LIN {X 0,Y 468.258,Z 232.885,A -85,B 0,C 180,E1 -7689.078,E2 -7689.078} C_VEL
LIN {X 0,Y 467.789,Z 228.961,A -85,B 0,C 180,E1 -7691.38,E2 -7691.38} C_VEL
LIN {X 0,Y 467.563,Z 227.872,A -85,B 0,C 180,E1 -7692.126,E2 -7692.126} C_VEL
LIN {X 0,Y 467.566,Z 227.872,A -85,B 0,C 180,E1 -7695.053,E2 -7695.053} C_VEL
LIN {X 0,Y 467.59,Z 227.868,A -85,B 0,C 180,E1 -7697.44,E2 -7697.44} C_VEL
LIN {X 0,Y 467.576,Z 227.87,A -85,B 0,C 180,E1 -7700.855,E2 -7700.855} C_VEL
LIN {X 0,Y 467.558,Z 227.874,A -85,B 0,C 180,E1 -7704.261,E2 -7704.261} C_VEL
LIN {X 0,Y 467.583,Z 227.869,A -85,B 0,C 180,E1 -7707.321,E2 -7707.321} C_VEL
LIN {X 0,Y 467.554,Z 227.872,A -85,B 0,C 180,E1 -7710.671,E2 -7710.671} C_VEL
LIN {X 0,Y 467.559,Z 227.867,A -85,B 0,C 180,E1 -7713.196,E2 -7713.196} C_VEL
LIN {X 0,Y 467.591,Z 227.864,A -85,B 0,C 180,E1 -7716.469,E2 -7716.469} C_VEL
LIN {X 0,Y 467.622,Z 227.86,A -85,B 0,C 180,E1 -7719.777,E2 -7719.777} C_VEL
LIN {X 0,Y 467.591,Z 227.864,A -85,B 0,C 180,E1 -7722.506,E2 -7722.506} C_VEL
LIN {X 0,Y 467.611,Z 227.864,A -85,B 0,C 180,E1 -7725.197,E2 -7725.197} C_VEL
LIN {X 0,Y 467.658,Z 227.855,A -85,B 0,C 180,E1 -7727.855,E2 -7727.855} C_VEL
LIN {X 0,Y 467.659,Z 227.855,A -85,B 0,C 180,E1 -7731.357,E2 -7731.357} C_VEL
LIN {X 0,Y 467.713,Z 227.849,A -85,B 0,C 180,E1 -7733.962,E2 -7733.962} C_VEL
LIN {X 0,Y 467.861,Z 227.83,A -85,B 0,C 180,E1 -7737.417,E2 -7737.417} C_VEL
LIN {X 0,Y 467.88,Z 227.832,A -85,B 0,C 180,E1 -7740,E2 -7740} C_VEL
LIN {X 0,Y 467.849,Z 227.831,A -85,B 0,C 180,E1 -7742.583,E2 -7742.583} C_VEL
LIN {X 0,Y 467.737,Z 227.846,A -85,B 0,C 180,E1 -7746.038,E2 -7746.038} C_VEL
LIN {X 0,Y 467.682,Z 227.852,A -85,B 0,C 180,E1 -7748.643,E2 -7748.643} C_VEL
LIN {X 0,Y 467.656,Z 227.855,A -85,B 0,C 180,E1 -7752.358,E2 -7752.358} C_VEL
LIN {X 0,Y 467.652,Z 227.858,A -85,B 0,C 180,E1 -7755.885,E2 -7755.885} C_VEL
LIN {X 0,Y 467.625,Z 227.863,A -85,B 0,C 180,E1 -7759.308,E2 -7759.308} C_VEL
LIN {X 0,Y 467.536,Z 227.87,A -85,B 0,C 180,E1 -7762.074,E2 -7762.074} C_VEL
LIN {X 0,Y 467.587,Z 227.864,A -85,B 0,C 180,E1 -7764.888,E2 -7764.888} C_VEL
LIN {X 0,Y 467.621,Z 227.863,A -85,B 0,C 180,E1 -7767.769,E2 -7767.769} C_VEL
LIN {X 0,Y 467.569,Z 227.869,A -85,B 0,C 180,E1 -7771.045,E2 -7771.045} C_VEL
LIN {X 0,Y 467.579,Z 227.868,A -85,B 0,C 180,E1 -7774.24,E2 -7774.24} C_VEL
LIN {X 0,Y 467.549,Z 227.873,A -85,B 0,C 180,E1 -7777.186,E2 -7777.186} C_VEL
LIN {X 0,Y 467.56,Z 227.869,A -85,B 0,C 180,E1 -7780.267,E2 -7780.267} C_VEL
LIN {X 0,Y 467.549,Z 227.874,A -85,B 0,C 180,E1 -7783.745,E2 -7783.745} C_VEL
LIN {X 0,Y 467.556,Z 227.869,A -85,B 0,C 180,E1 -7786.255,E2 -7786.255} C_VEL
LIN {X 0,Y 467.572,Z 227.872,A -85,B 0,C 180,E1 -7788.724,E2 -7788.724} C_VEL
LIN {X 0,Y 467.563,Z 227.872,A -85,B 0,C 180,E1 -7790.049,E2 -7790.049} C_VEL
LIN {X 0,Y 467.556,Z 228.203,A -85,B 0,C 180,E1 -7790.853,E2 -7790.853} C_VEL
LIN {X 0,Y 467.607,Z 231.102,A -85,B 0,C 180,E1 -7793.045,E2 -7793.045} C_VEL
LIN {X 0,Y 467.545,Z 234.837,A -85,B 0,C 180,E1 -7795.766,E2 -7795.766} C_VEL
LIN {X 0,Y 467.357,Z 239.771,A -85,B 0,C 180,E1 -7799.251,E2 -7799.251} C_VEL
LIN {X 0,Y 467.155,Z 244.635,A -85,B 0,C 180,E1 -7802.575,E2 -7802.575} C_VEL
LIN {X 0,Y 467.087,Z 248.387,A -85,B 0,C 180,E1 -7805.083,E2 -7805.083} C_VEL
LIN {X 0,Y 466.975,Z 252.771,A -85,B 0,C 180,E1 -7807.898,E2 -7807.898} C_VEL
LIN {X 0,Y 466.904,Z 258.071,A -85,B 0,C 180,E1 -7811.245,E2 -7811.245} C_VEL
LIN {X 0,Y 466.903,Z 258.381,A -85,B 0,C 180,E1 -7811.432,E2 -7811.432} C_VEL
LIN {X 0,Y 470.586,Z 273.156,A -85,B 0,C 180,E1 -7811.948,E2 -7811.948} C_VEL
LIN {X 0,Y 471.87,Z 279.673,A -85,B 0,C 180,E1 -7812.223,E2 -7812.223} C_VEL
LIN {X 0,Y 471.651,Z 287.48,A -85,B 0,C 180,E1 -7812.533,E2 -7812.533} C_VEL
LIN {X 0,Y 470.858,Z 293.031,A -85,B 0,C 180,E1 -7812.76,E2 -7812.76} C_VEL
LIN {X 0,Y 467.715,Z 301.937,A -85,B 0,C 180,E1 -7813.131,E2 -7813.131} C_VEL
LIN {X 0,Y 464.47,Z 310.546,A -85,B 0,C 180,E1 -7813.583,E2 -7813.583} C_VEL
LIN {X 0,Y 463.524,Z 315.627,A -85,B 0,C 180,E1 -7813.933,E2 -7813.933} C_VEL
LIN {X 0,Y 462.813,Z 327.365,A -85,B 0,C 180,E1 -7814.927,E2 -7814.927} C_VEL
LIN {X 0,Y 462.041,Z 339.043,A -85,B 0,C 180,E1 -7816.139,E2 -7816.139} C_VEL
LIN {X 0,Y 461.354,Z 349.678,A -85,B 0,C 180,E1 -7817.491,E2 -7817.491} C_VEL
LIN {X 0,Y 460.845,Z 358.072,A -85,B 0,C 180,E1 -7818.788,E2 -7818.788} C_VEL
LIN {X 0,Y 460.359,Z 366.316,A -85,B 0,C 180,E1 -7820.333,E2 -7820.333} C_VEL
LIN {X 0,Y 460.082,Z 372.056,A -85,B 0,C 180,E1 -7821.656,E2 -7821.656} C_VEL
LIN {X 0,Y 459.847,Z 376.778,A -85,B 0,C 180,E1 -7822.977,E2 -7822.977} C_VEL
LIN {X 0,Y 459.728,Z 381.668,A -85,B 0,C 180,E1 -7824.737,E2 -7824.737} C_VEL
LIN {X 0,Y 459.623,Z 385.073,A -85,B 0,C 180,E1 -7826.493,E2 -7826.493} C_VEL
LIN {X 0,Y 459.519,Z 387.099,A -85,B 0,C 180,E1 -7828.247,E2 -7828.247} C_VEL
LIN {X 0,Y 459.5,Z 387.796,A -85,B 0,C 180,E1 -7830,E2 -7830} C_VEL
LIN {X 0,Y 459.518,Z 387.175,A -85,B 0,C 180,E1 -7831.753,E2 -7831.753} C_VEL
LIN {X 0,Y 459.622,Z 385.219,A -85,B 0,C 180,E1 -7833.507,E2 -7833.507} C_VEL
LIN {X 0,Y 459.722,Z 381.883,A -85,B 0,C 180,E1 -7835.263,E2 -7835.263} C_VEL
LIN {X 0,Y 459.847,Z 377.072,A -85,B 0,C 180,E1 -7837.023,E2 -7837.023} C_VEL
LIN {X 0,Y 460.134,Z 370.627,A -85,B 0,C 180,E1 -7838.786,E2 -7838.786} C_VEL
LIN {X 0,Y 460.502,Z 363.45,A -85,B 0,C 180,E1 -7840.331,E2 -7840.331} C_VEL
LIN {X 0,Y 461.108,Z 354.57,A -85,B 0,C 180,E1 -7841.874,E2 -7841.874} C_VEL
LIN {X 0,Y 461.665,Z 345.24,A -85,B 0,C 180,E1 -7843.2,E2 -7843.2} C_VEL
LIN {X 0,Y 462.317,Z 334.904,A -85,B 0,C 180,E1 -7844.414,E2 -7844.414} C_VEL
LIN {X 0,Y 463.038,Z 323.496,A -85,B 0,C 180,E1 -7845.516,E2 -7845.516} C_VEL
LIN {X 0,Y 463.776,Z 310.849,A -85,B 0,C 180,E1 -7846.507,E2 -7846.507} C_VEL
LIN {X 0,Y 464.402,Z 297.961,A -85,B 0,C 180,E1 -7847.311,E2 -7847.311} C_VEL
LIN {X 0,Y 464.97,Z 283.959,A -85,B 0,C 180,E1 -7847.979,E2 -7847.979} C_VEL
LIN {X 0,Y 464.881,Z 279.458,A -85,B 0,C 180,E1 -7848.16,E2 -7848.16} C_VEL
LIN {X 0,Y 461.702,Z 265.746,A -85,B 0,C 180,E1 -7848.721,E2 -7848.721} C_VEL
LIN {X 0,Y 459.856,Z 258.473,A -85,B 0,C 180,E1 -7848.975,E2 -7848.975} C_VEL
LIN {X 0,Y 459.938,Z 253.029,A -85,B 0,C 180,E1 -7852.458,E2 -7852.458} C_VEL
LIN {X 0,Y 460.035,Z 248.128,A -85,B 0,C 180,E1 -7855.664,E2 -7855.664} C_VEL
LIN {X 0,Y 460.143,Z 244.325,A -85,B 0,C 180,E1 -7858.261,E2 -7858.261} C_VEL
LIN {X 0,Y 460.332,Z 240.017,A -85,B 0,C 180,E1 -7861.271,E2 -7861.271} C_VEL
LIN {X 0,Y 460.526,Z 235.502,A -85,B 0,C 180,E1 -7864.504,E2 -7864.504} C_VEL
LIN {X 0,Y 460.553,Z 231.318,A -85,B 0,C 180,E1 -7867.618,E2 -7867.618} C_VEL
LIN {X 0,Y 460.542,Z 229.642,A -85,B 0,C 180,E1 -7868.897,E2 -7868.897} C_VEL
LIN {X 0,Y 460.491,Z 228.756,A -85,B 0,C 180,E1 -7869.867,E2 -7869.867} C_VEL
LIN {X 0,Y 460.516,Z 228.749,A -85,B 0,C 180,E1 -7872.901,E2 -7872.901} C_VEL
LIN {X 0,Y 460.51,Z 228.748,A -85,B 0,C 180,E1 -7875.831,E2 -7875.831} C_VEL
LIN {X 0,Y 460.521,Z 228.746,A -85,B 0,C 180,E1 -7878.987,E2 -7878.987} C_VEL
LIN {X 0,Y 460.517,Z 228.749,A -85,B 0,C 180,E1 -7881.266,E2 -7881.266} C_VEL
LIN {X 0,Y 460.511,Z 228.749,A -85,B 0,C 180,E1 -7884.554,E2 -7884.554} C_VEL
LIN {X 0,Y 460.532,Z 228.747,A -85,B 0,C 180,E1 -7887.716,E2 -7887.716} C_VEL
LIN {X 0,Y 460.54,Z 228.746,A -85,B 0,C 180,E1 -7890.769,E2 -7890.769} C_VEL
LIN {X 0,Y 460.559,Z 228.741,A -85,B 0,C 180,E1 -7893.734,E2 -7893.734} C_VEL
LIN {X 0,Y 460.548,Z 228.741,A -85,B 0,C 180,E1 -7896.624,E2 -7896.624} C_VEL
LIN {X 0,Y 460.554,Z 228.74,A -85,B 0,C 180,E1 -7899.453,E2 -7899.453} C_VEL
LIN {X 0,Y 460.551,Z 228.744,A -85,B 0,C 180,E1 -7902.23,E2 -7902.23} C_VEL
LIN {X 0,Y 460.567,Z 228.739,A -85,B 0,C 180,E1 -7904.965,E2 -7904.965} C_VEL
LIN {X 0,Y 460.613,Z 228.736,A -85,B 0,C 180,E1 -7908.559,E2 -7908.559} C_VEL
LIN {X 0,Y 460.622,Z 228.731,A -85,B 0,C 180,E1 -7911.224,E2 -7911.224} C_VEL
LIN {X 0,Y 460.703,Z 228.723,A -85,B 0,C 180,E1 -7913.87,E2 -7913.87} C_VEL
LIN {X 0,Y 460.792,Z 228.71,A -85,B 0,C 180,E1 -7917.377,E2 -7917.377} C_VEL
LIN {X 0,Y 460.825,Z 228.71,A -85,B 0,C 180,E1 -7920,E2 -7920} C_VEL
LIN {X 0,Y 460.803,Z 228.708,A -85,B 0,C 180,E1 -7922.622,E2 -7922.622} C_VEL
LIN {X 0,Y 460.679,Z 228.726,A -85,B 0,C 180,E1 -7926.13,E2 -7926.13} C_VEL
LIN {X 0,Y 460.612,Z 228.733,A -85,B 0,C 180,E1 -7928.776,E2 -7928.776} C_VEL
LIN {X 0,Y 460.617,Z 228.732,A -85,B 0,C 180,E1 -7932.445,E2 -7932.445} C_VEL
LIN {X 0,Y 460.604,Z 228.737,A -85,B 0,C 180,E1 -7935.997,E2 -7935.997} C_VEL
LIN {X 0,Y 460.569,Z 228.743,A -85,B 0,C 180,E1 -7939.615,E2 -7939.615} C_VEL
LIN {X 0,Y 460.514,Z 228.747,A -85,B 0,C 180,E1 -7942.428,E2 -7942.428} C_VEL
LIN {X 0,Y 460.546,Z 228.742,A -85,B 0,C 180,E1 -7945.796,E2 -7945.796} C_VEL
LIN {X 0,Y 460.522,Z 228.748,A -85,B 0,C 180,E1 -7949.232,E2 -7949.232} C_VEL
LIN {X 0,Y 460.534,Z 228.746,A -85,B 0,C 180,E1 -7952.284,E2 -7952.284} C_VEL
LIN {X 0,Y 460.51,Z 228.75,A -85,B 0,C 180,E1 -7955.446,E2 -7955.446} C_VEL
LIN {X 0,Y 460.542,Z 228.747,A -85,B 0,C 180,E1 -7958.897,E2 -7958.897} C_VEL
LIN {X 0,Y 460.525,Z 228.751,A -85,B 0,C 180,E1 -7962.181,E2 -7962.181} C_VEL
LIN {X 0,Y 460.513,Z 228.751,A -85,B 0,C 180,E1 -7965.411,E2 -7965.411} C_VEL
LIN {X 0,Y 460.558,Z 228.925,A -85,B 0,C 180,E1 -7967.822,E2 -7967.822} C_VEL
LIN {X 0,Y 461.132,Z 232.835,A -85,B 0,C 180,E1 -7970.2,E2 -7970.2} C_VEL
LIN {X 0,Y 461.314,Z 236.792,A -85,B 0,C 180,E1 -7972.454,E2 -7972.454} C_VEL
LIN {X 0,Y 461.036,Z 242.718,A -85,B 0,C 180,E1 -7975.665,E2 -7975.665} C_VEL
LIN {X 0,Y 460.839,Z 248.673,A -85,B 0,C 180,E1 -7978.767,E2 -7978.767} C_VEL
LIN {X 0,Y 460.613,Z 255.61,A -85,B 0,C 180,E1 -7982.247,E2 -7982.247} C_VEL
LIN {X 0,Y 460.218,Z 262.588,A -85,B 0,C 180,E1 -7985.649,E2 -7985.649} C_VEL
LIN {X 0,Y 460.068,Z 268.978,A -85,B 0,C 180,E1 -7988.723,E2 -7988.723} C_VEL
LIN {X 0,Y 459.911,Z 273.938,A -85,B 0,C 180,E1 -7991.062,E2 -7991.062} C_VEL
LIN {X 0,Y 463.398,Z 290.247,A -85,B 0,C 180,E1 -7991.618,E2 -7991.618} C_VEL
LIN {X 0,Y 464.84,Z 299.475,A -85,B 0,C 180,E1 -7992.006,E2 -7992.006} C_VEL
LIN {X 0,Y 464.311,Z 313.432,A -85,B 0,C 180,E1 -7992.653,E2 -7992.653} C_VEL
LIN {X 0,Y 463.49,Z 327.092,A -85,B 0,C 180,E1 -7993.482,E2 -7993.482} C_VEL
LIN {X 0,Y 462.776,Z 339.91,A -85,B 0,C 180,E1 -7994.475,E2 -7994.475} C_VEL
LIN {X 0,Y 462.063,Z 351.466,A -85,B 0,C 180,E1 -7995.578,E2 -7995.578} C_VEL
LIN {X 0,Y 461.426,Z 361.937,A -85,B 0,C 180,E1 -7996.793,E2 -7996.793} C_VEL
LIN {X 0,Y 460.914,Z 371.401,A -85,B 0,C 180,E1 -7998.121,E2 -7998.121} C_VEL
LIN {X 0,Y 460.319,Z 380.415,A -85,B 0,C 180,E1 -7999.665,E2 -7999.665} C_VEL
LIN {X 0,Y 459.98,Z 387.7,A -85,B 0,C 180,E1 -8001.211,E2 -8001.211} C_VEL
LIN {X 0,Y 459.738,Z 394.247,A -85,B 0,C 180,E1 -8002.975,E2 -8002.975} C_VEL
LIN {X 0,Y 459.645,Z 399.148,A -85,B 0,C 180,E1 -8004.736,E2 -8004.736} C_VEL
LIN {X 0,Y 459.547,Z 402.554,A -85,B 0,C 180,E1 -8006.493,E2 -8006.493} C_VEL
LIN {X 0,Y 459.514,Z 404.57,A -85,B 0,C 180,E1 -8008.247,E2 -8008.247} C_VEL
LIN {X 0,Y 459.499,Z 405.238,A -85,B 0,C 180,E1 -8010,E2 -8010} C_VEL
LIN {X 0,Y 459.514,Z 404.571,A -85,B 0,C 180,E1 -8011.753,E2 -8011.753} C_VEL
LIN {X 0,Y 459.547,Z 402.558,A -85,B 0,C 180,E1 -8013.507,E2 -8013.507} C_VEL
LIN {X 0,Y 459.644,Z 399.15,A -85,B 0,C 180,E1 -8015.264,E2 -8015.264} C_VEL
LIN {X 0,Y 459.734,Z 394.243,A -85,B 0,C 180,E1 -8017.025,E2 -8017.025} C_VEL
LIN {X 0,Y 459.98,Z 387.696,A -85,B 0,C 180,E1 -8018.789,E2 -8018.789} C_VEL
LIN {X 0,Y 460.319,Z 380.412,A -85,B 0,C 180,E1 -8020.334,E2 -8020.334} C_VEL
LIN {X 0,Y 460.891,Z 371.394,A -85,B 0,C 180,E1 -8021.88,E2 -8021.88} C_VEL
LIN {X 0,Y 461.425,Z 361.929,A -85,B 0,C 180,E1 -8023.207,E2 -8023.207} C_VEL
LIN {X 0,Y 462.046,Z 351.452,A -85,B 0,C 180,E1 -8024.423,E2 -8024.423} C_VEL
LIN {X 0,Y 462.743,Z 339.894,A -85,B 0,C 180,E1 -8025.526,E2 -8025.526} C_VEL
LIN {X 0,Y 463.496,Z 327.074,A -85,B 0,C 180,E1 -8026.517,E2 -8026.517} C_VEL
LIN {X 0,Y 464.277,Z 314.068,A -85,B 0,C 180,E1 -8027.31,E2 -8027.31} C_VEL
LIN {X 0,Y 464.801,Z 300.72,A -85,B 0,C 180,E1 -8027.939,E2 -8027.939} C_VEL
LIN {X 0,Y 464.292,Z 295.229,A -85,B 0,C 180,E1 -8028.173,E2 -8028.173} C_VEL
LIN {X 0,Y 461.513,Z 281.294,A -85,B 0,C 180,E1 -8028.708,E2 -8028.708} C_VEL
LIN {X 0,Y 459.913,Z 273.921,A -85,B 0,C 180,E1 -8028.941,E2 -8028.941} C_VEL
LIN {X 0,Y 460.069,Z 268.49,A -85,B 0,C 180,E1 -8031.508,E2 -8031.508} C_VEL
LIN {X 0,Y 460.214,Z 262.58,A -85,B 0,C 180,E1 -8034.351,E2 -8034.351} C_VEL
LIN {X 0,Y 460.611,Z 255.593,A -85,B 0,C 180,E1 -8037.753,E2 -8037.753} C_VEL
LIN {X 0,Y 460.804,Z 248.443,A -85,B 0,C 180,E1 -8041.341,E2 -8041.341} C_VEL
LIN {X 0,Y 461.08,Z 242.189,A -85,B 0,C 180,E1 -8044.604,E2 -8044.604} C_VEL
LIN {X 0,Y 461.312,Z 236.658,A -85,B 0,C 180,E1 -8047.607,E2 -8047.607} C_VEL
LIN {X 0,Y 461.131,Z 232.825,A -85,B 0,C 180,E1 -8049.8,E2 -8049.8} C_VEL
LIN {X 0,Y 460.525,Z 228.748,A -85,B 0,C 180,E1 -8052.32,E2 -8052.32} C_VEL
LIN {X 0,Y 460.514,Z 228.75,A -85,B 0,C 180,E1 -8055.411,E2 -8055.411} C_VEL
LIN {X 0,Y 460.533,Z 228.744,A -85,B 0,C 180,E1 -8058.398,E2 -8058.398} C_VEL
LIN {X 0,Y 460.523,Z 228.749,A -85,B 0,C 180,E1 -8061.267,E2 -8061.267} C_VEL
LIN {X 0,Y 460.509,Z 228.75,A -85,B 0,C 180,E1 -8064.554,E2 -8064.554} C_VEL
LIN {X 0,Y 460.533,Z 228.747,A -85,B 0,C 180,E1 -8067.716,E2 -8067.716} C_VEL
LIN {X 0,Y 460.524,Z 228.749,A -85,B 0,C 180,E1 -8070.768,E2 -8070.768} C_VEL
LIN {X 0,Y 460.528,Z 228.745,A -85,B 0,C 180,E1 -8073.733,E2 -8073.733} C_VEL
LIN {X 0,Y 460.545,Z 228.742,A -85,B 0,C 180,E1 -8076.624,E2 -8076.624} C_VEL
LIN {X 0,Y 460.552,Z 228.741,A -85,B 0,C 180,E1 -8079.453,E2 -8079.453} C_VEL
LIN {X 0,Y 460.544,Z 228.744,A -85,B 0,C 180,E1 -8082.23,E2 -8082.23} C_VEL
LIN {X 0,Y 460.569,Z 228.739,A -85,B 0,C 180,E1 -8084.965,E2 -8084.965} C_VEL
LIN {X 0,Y 460.612,Z 228.736,A -85,B 0,C 180,E1 -8088.559,E2 -8088.559} C_VEL
LIN {X 0,Y 460.611,Z 228.733,A -85,B 0,C 180,E1 -8091.224,E2 -8091.224} C_VEL
LIN {X 0,Y 460.678,Z 228.726,A -85,B 0,C 180,E1 -8093.87,E2 -8093.87} C_VEL
LIN {X 0,Y 460.802,Z 228.709,A -85,B 0,C 180,E1 -8097.378,E2 -8097.378} C_VEL
LIN {X 0,Y 460.85,Z 228.708,A -85,B 0,C 180,E1 -8100,E2 -8100} C_VEL
LIN {X 0,Y 460.79,Z 228.711,A -85,B 0,C 180,E1 -8102.623,E2 -8102.623} C_VEL
LIN {X 0,Y 460.703,Z 228.723,A -85,B 0,C 180,E1 -8106.13,E2 -8106.13} C_VEL
LIN {X 0,Y 460.629,Z 228.73,A -85,B 0,C 180,E1 -8108.776,E2 -8108.776} C_VEL
LIN {X 0,Y 460.599,Z 228.735,A -85,B 0,C 180,E1 -8112.435,E2 -8112.435} C_VEL
LIN {X 0,Y 460.602,Z 228.737,A -85,B 0,C 180,E1 -8115.998,E2 -8115.998} C_VEL
LIN {X 0,Y 460.573,Z 228.738,A -85,B 0,C 180,E1 -8118.902,E2 -8118.902} C_VEL
LIN {X 0,Y 460.518,Z 228.745,A -85,B 0,C 180,E1 -8121.486,E2 -8121.486} C_VEL
LIN {X 0,Y 460.533,Z 228.747,A -85,B 0,C 180,E1 -8124.333,E2 -8124.333} C_VEL
LIN {X 0,Y 460.573,Z 228.739,A -85,B 0,C 180,E1 -8127.244,E2 -8127.244} C_VEL
LIN {X 0,Y 460.512,Z 228.746,A -85,B 0,C 180,E1 -8130.24,E2 -8130.24} C_VEL
LIN {X 0,Y 460.521,Z 228.744,A -85,B 0,C 180,E1 -8133.326,E2 -8133.326} C_VEL
LIN {X 0,Y 460.478,Z 228.75,A -85,B 0,C 180,E1 -8136.529,E2 -8136.529} C_VEL
LIN {X 0,Y 460.514,Z 228.745,A -85,B 0,C 180,E1 -8139.864,E2 -8139.864} C_VEL
LIN {X 0,Y 460.48,Z 228.751,A -85,B 0,C 180,E1 -8142.896,E2 -8142.896} C_VEL
LIN {X 0,Y 460.51,Z 228.748,A -85,B 0,C 180,E1 -8145.831,E2 -8145.831} C_VEL
LIN {X 0,Y 460.524,Z 228.748,A -85,B 0,C 180,E1 -8148.988,E2 -8148.988} C_VEL
LIN {X 0,Y 460.508,Z 228.75,A -85,B 0,C 180,E1 -8150.135,E2 -8150.135} C_VEL
LIN {X 0,Y 460.553,Z 229.73,A -85,B 0,C 180,E1 -8151.27,E2 -8151.27} C_VEL
LIN {X 0,Y 460.534,Z 234.083,A -85,B 0,C 180,E1 -8154.556,E2 -8154.556} C_VEL
LIN {X 0,Y 460.396,Z 237.578,A -85,B 0,C 180,E1 -8157.096,E2 -8157.096} C_VEL
LIN {X 0,Y 460.251,Z 241.31,A -85,B 0,C 180,E1 -8159.741,E2 -8159.741} C_VEL
LIN {X 0,Y 460.082,Z 245.618,A -85,B 0,C 180,E1 -8162.725,E2 -8162.725} C_VEL
LIN {X 0,Y 460.008,Z 249.964,A -85,B 0,C 180,E1 -8165.638,E2 -8165.638} C_VEL
LIN {X 0,Y 459.907,Z 254.8,A -85,B 0,C 180,E1 -8168.775,E2 -8168.775} C_VEL
LIN {X 0,Y 459.855,Z 258.498,A -85,B 0,C 180,E1 -8171.134,E2 -8171.134} C_VEL
LIN {X 0,Y 463.604,Z 273.574,A -85,B 0,C 180,E1 -8171.674,E2 -8171.674} C_VEL
LIN {X 0,Y 465.08,Z 281.025,A -85,B 0,C 180,E1 -8171.999,E2 -8171.999} C_VEL
LIN {X 0,Y 464.612,Z 293.881,A -85,B 0,C 180,E1 -8172.566,E2 -8172.566} C_VEL
LIN {X 0,Y 463.991,Z 306.273,A -85,B 0,C 180,E1 -8173.274,E2 -8173.274} C_VEL
LIN {X 0,Y 463.524,Z 315.627,A -85,B 0,C 180,E1 -8173.933,E2 -8173.933} C_VEL
LIN {X 0,Y 462.588,Z 320.688,A -85,B 0,C 180,E1 -8174.312,E2 -8174.312} C_VEL
LIN {X 0,Y 459.314,Z 328.655,A -85,B 0,C 180,E1 -8174.928,E2 -8174.928} C_VEL
LIN {X 0,Y 456.014,Z 336.214,A -85,B 0,C 180,E1 -8175.606,E2 -8175.606} C_VEL
LIN {X 0,Y 455.014,Z 340.561,A -85,B 0,C 180,E1 -8176.084,E2 -8176.084} C_VEL
LIN {X 0,Y 454.364,Z 350.101,A -85,B 0,C 180,E1 -8177.335,E2 -8177.335} C_VEL
LIN {X 0,Y 453.866,Z 358.21,A -85,B 0,C 180,E1 -8178.613,E2 -8178.613} C_VEL
LIN {X 0,Y 453.35,Z 366.453,A -85,B 0,C 180,E1 -8180.182,E2 -8180.182} C_VEL
LIN {X 0,Y 453.046,Z 372.193,A -85,B 0,C 180,E1 -8181.525,E2 -8181.525} C_VEL
LIN {X 0,Y 452.772,Z 376.915,A -85,B 0,C 180,E1 -8182.867,E2 -8182.867} C_VEL
LIN {X 0,Y 452.671,Z 381.804,A -85,B 0,C 180,E1 -8184.655,E2 -8184.655} C_VEL
LIN {X 0,Y 452.522,Z 385.209,A -85,B 0,C 180,E1 -8186.438,E2 -8186.438} C_VEL
LIN {X 0,Y 452.435,Z 387.233,A -85,B 0,C 180,E1 -8188.22,E2 -8188.22} C_VEL
LIN {X 0,Y 452.406,Z 387.931,A -85,B 0,C 180,E1 -8190,E2 -8190} C_VEL
LIN {X 0,Y 452.434,Z 387.309,A -85,B 0,C 180,E1 -8191.78,E2 -8191.78} C_VEL
LIN {X 0,Y 452.521,Z 385.353,A -85,B 0,C 180,E1 -8193.562,E2 -8193.562} C_VEL
LIN {X 0,Y 452.661,Z 382.017,A -85,B 0,C 180,E1 -8195.345,E2 -8195.345} C_VEL
LIN {X 0,Y 452.771,Z 377.206,A -85,B 0,C 180,E1 -8197.133,E2 -8197.133} C_VEL
LIN {X 0,Y 453.097,Z 370.76,A -85,B 0,C 180,E1 -8198.923,E2 -8198.923} C_VEL
LIN {X 0,Y 453.49,Z 363.583,A -85,B 0,C 180,E1 -8200.492,E2 -8200.492} C_VEL
LIN {X 0,Y 454.144,Z 354.702,A -85,B 0,C 180,E1 -8202.059,E2 -8202.059} C_VEL
LIN {X 0,Y 454.729,Z 345.372,A -85,B 0,C 180,E1 -8203.405,E2 -8203.405} C_VEL
LIN {X 0,Y 455.421,Z 335.035,A -85,B 0,C 180,E1 -8204.637,E2 -8204.637} C_VEL
LIN {X 0,Y 456.169,Z 323.626,A -85,B 0,C 180,E1 -8205.756,E2 -8205.756} C_VEL
LIN {X 0,Y 456.974,Z 310.977,A -85,B 0,C 180,E1 -8206.76,E2 -8206.76} C_VEL
LIN {X 0,Y 457.662,Z 297.481,A -85,B 0,C 180,E1 -8207.61,E2 -8207.61} C_VEL
LIN {X 0,Y 458.222,Z 284.087,A -85,B 0,C 180,E1 -8208.253,E2 -8208.253} C_VEL
LIN {X 0,Y 458.026,Z 280.182,A -85,B 0,C 180,E1 -8208.419,E2 -8208.419} C_VEL
LIN {X 0,Y 455.012,Z 267.307,A -85,B 0,C 180,E1 -8208.969,E2 -8208.969} C_VEL
LIN {X 0,Y 452.768,Z 258.605,A -85,B 0,C 180,E1 -8209.284,E2 -8209.284} C_VEL
LIN {X 0,Y 452.84,Z 254.619,A -85,B 0,C 180,E1 -8211.869,E2 -8211.869} C_VEL
LIN {X 0,Y 452.954,Z 250.218,A -85,B 0,C 180,E1 -8214.767,E2 -8214.767} C_VEL
LIN {X 0,Y 453.058,Z 245.707,A -85,B 0,C 180,E1 -8217.846,E2 -8217.846} C_VEL
LIN {X 0,Y 453.244,Z 241.543,A -85,B 0,C 180,E1 -8220.777,E2 -8220.777} C_VEL
LIN {X 0,Y 453.412,Z 237.208,A -85,B 0,C 180,E1 -8223.918,E2 -8223.918} C_VEL
LIN {X 0,Y 453.507,Z 233.991,A -85,B 0,C 180,E1 -8226.308,E2 -8226.308} C_VEL
LIN {X 0,Y 453.447,Z 229.92,A -85,B 0,C 180,E1 -8229.455,E2 -8229.455} C_VEL
LIN {X 0,Y 453.476,Z 229.624,A -85,B 0,C 180,E1 -8231.934,E2 -8231.934} C_VEL
LIN {X 0,Y 453.488,Z 229.622,A -85,B 0,C 180,E1 -8235.471,E2 -8235.471} C_VEL
LIN {X 0,Y 453.455,Z 229.628,A -85,B 0,C 180,E1 -8238.206,E2 -8238.206} C_VEL
LIN {X 0,Y 453.468,Z 229.625,A -85,B 0,C 180,E1 -8240.798,E2 -8240.798} C_VEL
LIN {X 0,Y 453.457,Z 229.626,A -85,B 0,C 180,E1 -8243.917,E2 -8243.917} C_VEL
LIN {X 0,Y 453.481,Z 229.622,A -85,B 0,C 180,E1 -8247.151,E2 -8247.151} C_VEL
LIN {X 0,Y 453.475,Z 229.622,A -85,B 0,C 180,E1 -8250.268,E2 -8250.268} C_VEL
LIN {X 0,Y 453.505,Z 229.618,A -85,B 0,C 180,E1 -8253.294,E2 -8253.294} C_VEL
LIN {X 0,Y 453.501,Z 229.62,A -85,B 0,C 180,E1 -8256.239,E2 -8256.239} C_VEL
LIN {X 0,Y 453.486,Z 229.624,A -85,B 0,C 180,E1 -8259.118,E2 -8259.118} C_VEL
LIN {X 0,Y 453.505,Z 229.62,A -85,B 0,C 180,E1 -8261.944,E2 -8261.944} C_VEL
LIN {X 0,Y 453.542,Z 229.613,A -85,B 0,C 180,E1 -8264.726,E2 -8264.726} C_VEL
LIN {X 0,Y 453.562,Z 229.613,A -85,B 0,C 180,E1 -8268.379,E2 -8268.379} C_VEL
LIN {X 0,Y 453.588,Z 229.608,A -85,B 0,C 180,E1 -8271.086,E2 -8271.086} C_VEL
LIN {X 0,Y 453.67,Z 229.6,A -85,B 0,C 180,E1 -8273.775,E2 -8273.775} C_VEL
LIN {X 0,Y 453.736,Z 229.589,A -85,B 0,C 180,E1 -8277.337,E2 -8277.337} C_VEL
LIN {X 0,Y 453.795,Z 229.586,A -85,B 0,C 180,E1 -8280,E2 -8280} C_VEL
LIN {X 0,Y 453.747,Z 229.587,A -85,B 0,C 180,E1 -8282.663,E2 -8282.663} C_VEL
LIN {X 0,Y 453.645,Z 229.603,A -85,B 0,C 180,E1 -8286.226,E2 -8286.226} C_VEL
LIN {X 0,Y 453.58,Z 229.609,A -85,B 0,C 180,E1 -8288.914,E2 -8288.914} C_VEL
LIN {X 0,Y 453.567,Z 229.611,A -85,B 0,C 180,E1 -8292.529,E2 -8292.529} C_VEL
LIN {X 0,Y 453.547,Z 229.618,A -85,B 0,C 180,E1 -8296.196,E2 -8296.196} C_VEL
LIN {X 0,Y 453.519,Z 229.617,A -85,B 0,C 180,E1 -8299.039,E2 -8299.039} C_VEL
LIN {X 0,Y 453.479,Z 229.622,A -85,B 0,C 180,E1 -8301.836,E2 -8301.836} C_VEL
LIN {X 0,Y 453.497,Z 229.619,A -85,B 0,C 180,E1 -8304.735,E2 -8304.735} C_VEL
LIN {X 0,Y 453.465,Z 229.625,A -85,B 0,C 180,E1 -8307.943,E2 -8307.943} C_VEL
LIN {X 0,Y 453.476,Z 229.626,A -85,B 0,C 180,E1 -8310.76,E2 -8310.76} C_VEL
LIN {X 0,Y 453.479,Z 229.625,A -85,B 0,C 180,E1 -8313.913,E2 -8313.913} C_VEL
LIN {X 0,Y 453.451,Z 229.631,A -85,B 0,C 180,E1 -8317.19,E2 -8317.19} C_VEL
LIN {X 0,Y 453.488,Z 229.622,A -85,B 0,C 180,E1 -8319.45,E2 -8319.45} C_VEL
LIN {X 0,Y 453.478,Z 229.626,A -85,B 0,C 180,E1 -8321.935,E2 -8321.935} C_VEL
LIN {X 0,Y 453.483,Z 229.626,A -85,B 0,C 180,E1 -8325.471,E2 -8325.471} C_VEL
LIN {X 0,Y 453.505,Z 229.773,A -85,B 0,C 180,E1 -8327.565,E2 -8327.565} C_VEL
LIN {X 0,Y 453.993,Z 232.781,A -85,B 0,C 180,E1 -8329.445,E2 -8329.445} C_VEL
LIN {X 0,Y 454.305,Z 236.716,A -85,B 0,C 180,E1 -8331.772,E2 -8331.772} C_VEL
LIN {X 0,Y 454.129,Z 240.663,A -85,B 0,C 180,E1 -8333.979,E2 -8333.979} C_VEL
LIN {X 0,Y 453.88,Z 246.605,A -85,B 0,C 180,E1 -8337.183,E2 -8337.183} C_VEL
LIN {X 0,Y 453.67,Z 252.563,A -85,B 0,C 180,E1 -8340.282,E2 -8340.282} C_VEL
LIN {X 0,Y 453.559,Z 256.546,A -85,B 0,C 180,E1 -8342.299,E2 -8342.299} C_VEL
LIN {X 0,Y 453.166,Z 264.447,A -85,B 0,C 180,E1 -8346.22,E2 -8346.22} C_VEL
LIN {X 0,Y 452.967,Z 270.341,A -85,B 0,C 180,E1 -8349.093,E2 -8349.093} C_VEL
LIN {X 0,Y 452.828,Z 273.851,A -85,B 0,C 180,E1 -8350.763,E2 -8350.763} C_VEL
LIN {X 0,Y 456.057,Z 288.568,A -85,B 0,C 180,E1 -8351.262,E2 -8351.262} C_VEL
LIN {X 0,Y 458.045,Z 299.839,A -85,B 0,C 180,E1 -8351.751,E2 -8351.751} C_VEL
LIN {X 0,Y 457.516,Z 313.508,A -85,B 0,C 180,E1 -8352.399,E2 -8352.399} C_VEL
LIN {X 0,Y 456.673,Z 326.96,A -85,B 0,C 180,E1 -8353.228,E2 -8353.228} C_VEL
LIN {X 0,Y 455.9,Z 339.777,A -85,B 0,C 180,E1 -8354.234,E2 -8354.234} C_VEL
LIN {X 0,Y 455.146,Z 351.333,A -85,B 0,C 180,E1 -8355.354,E2 -8355.354} C_VEL
LIN {X 0,Y 454.475,Z 361.804,A -85,B 0,C 180,E1 -8356.587,E2 -8356.587} C_VEL
LIN {X 0,Y 453.904,Z 371.267,A -85,B 0,C 180,E1 -8357.935,E2 -8357.935} C_VEL
LIN {X 0,Y 453.299,Z 380.281,A -85,B 0,C 180,E1 -8359.504,E2 -8359.504} C_VEL
LIN {X 0,Y 452.929,Z 387.565,A -85,B 0,C 180,E1 -8361.073,E2 -8361.073} C_VEL
LIN {X 0,Y 452.664,Z 394.112,A -85,B 0,C 180,E1 -8362.865,E2 -8362.865} C_VEL
LIN {X 0,Y 452.559,Z 399.013,A -85,B 0,C 180,E1 -8364.654,E2 -8364.654} C_VEL
LIN {X 0,Y 452.445,Z 402.42,A -85,B 0,C 180,E1 -8366.438,E2 -8366.438} C_VEL
LIN {X 0,Y 452.43,Z 404.436,A -85,B 0,C 180,E1 -8368.22,E2 -8368.22} C_VEL
LIN {X 0,Y 452.405,Z 405.104,A -85,B 0,C 180,E1 -8370,E2 -8370} C_VEL
LIN {X 0,Y 452.43,Z 404.436,A -85,B 0,C 180,E1 -8371.78,E2 -8371.78} C_VEL
LIN {X 0,Y 452.445,Z 402.422,A -85,B 0,C 180,E1 -8373.562,E2 -8373.562} C_VEL
LIN {X 0,Y 452.558,Z 399.014,A -85,B 0,C 180,E1 -8375.346,E2 -8375.346} C_VEL
LIN {X 0,Y 452.661,Z 394.107,A -85,B 0,C 180,E1 -8377.135,E2 -8377.135} C_VEL
LIN {X 0,Y 452.929,Z 387.56,A -85,B 0,C 180,E1 -8378.926,E2 -8378.926} C_VEL
LIN {X 0,Y 453.299,Z 380.275,A -85,B 0,C 180,E1 -8380.496,E2 -8380.496} C_VEL
LIN {X 0,Y 453.887,Z 371.256,A -85,B 0,C 180,E1 -8382.066,E2 -8382.066} C_VEL
LIN {X 0,Y 454.475,Z 361.791,A -85,B 0,C 180,E1 -8383.412,E2 -8383.412} C_VEL
LIN {X 0,Y 455.145,Z 351.315,A -85,B 0,C 180,E1 -8384.646,E2 -8384.646} C_VEL
LIN {X 0,Y 455.883,Z 339.756,A -85,B 0,C 180,E1 -8385.766,E2 -8385.766} C_VEL
LIN {X 0,Y 456.673,Z 326.935,A -85,B 0,C 180,E1 -8386.771,E2 -8386.771} C_VEL
LIN {X 0,Y 457.494,Z 313.784,A -85,B 0,C 180,E1 -8387.583,E2 -8387.583} C_VEL
LIN {X 0,Y 458.026,Z 300.833,A -85,B 0,C 180,E1 -8388.203,E2 -8388.203} C_VEL
LIN {X 0,Y 456.621,Z 291.436,A -85,B 0,C 180,E1 -8388.62,E2 -8388.62} C_VEL
LIN {X 0,Y 453.581,Z 277.233,A -85,B 0,C 180,E1 -8389.135,E2 -8389.135} C_VEL
LIN {X 0,Y 452.836,Z 273.765,A -85,B 0,C 180,E1 -8389.261,E2 -8389.261} C_VEL
LIN {X 0,Y 452.997,Z 268.366,A -85,B 0,C 180,E1 -8391.86,E2 -8391.86} C_VEL
LIN {X 0,Y 453.16,Z 262.466,A -85,B 0,C 180,E1 -8394.755,E2 -8394.755} C_VEL
LIN {X 0,Y 453.562,Z 256.001,A -85,B 0,C 180,E1 -8397.967,E2 -8397.967} C_VEL
LIN {X 0,Y 453.701,Z 250.548,A -85,B 0,C 180,E1 -8400.743,E2 -8400.743} C_VEL
LIN {X 0,Y 453.962,Z 244.592,A -85,B 0,C 180,E1 -8403.872,E2 -8403.872} C_VEL
LIN {X 0,Y 454.252,Z 238.671,A -85,B 0,C 180,E1 -8407.113,E2 -8407.113} C_VEL
LIN {X 0,Y 454.213,Z 234.733,A -85,B 0,C 180,E1 -8409.375,E2 -8409.375} C_VEL
LIN {X 0,Y 453.653,Z 230.505,A -85,B 0,C 180,E1 -8411.96,E2 -8411.96} C_VEL
LIN {X 0,Y 453.471,Z 229.627,A -85,B 0,C 180,E1 -8412.578,E2 -8412.578} C_VEL
LIN {X 0,Y 453.464,Z 229.629,A -85,B 0,C 180,E1 -8415.779,E2 -8415.779} C_VEL
LIN {X 0,Y 453.48,Z 229.624,A -85,B 0,C 180,E1 -8418.209,E2 -8418.209} C_VEL
LIN {X 0,Y 453.492,Z 229.624,A -85,B 0,C 180,E1 -8420.794,E2 -8420.794} C_VEL
LIN {X 0,Y 453.452,Z 229.628,A -85,B 0,C 180,E1 -8423.917,E2 -8423.917} C_VEL
LIN {X 0,Y 453.484,Z 229.624,A -85,B 0,C 180,E1 -8427.151,E2 -8427.151} C_VEL
LIN {X 0,Y 453.466,Z 229.624,A -85,B 0,C 180,E1 -8430.268,E2 -8430.268} C_VEL
LIN {X 0,Y 453.468,Z 229.623,A -85,B 0,C 180,E1 -8433.292,E2 -8433.292} C_VEL
LIN {X 0,Y 453.495,Z 229.62,A -85,B 0,C 180,E1 -8436.238,E2 -8436.238} C_VEL
LIN {X 0,Y 453.484,Z 229.624,A -85,B 0,C 180,E1 -8439.118,E2 -8439.118} C_VEL
LIN {X 0,Y 453.5,Z 229.622,A -85,B 0,C 180,E1 -8441.944,E2 -8441.944} C_VEL
LIN {X 0,Y 453.543,Z 229.613,A -85,B 0,C 180,E1 -8444.726,E2 -8444.726} C_VEL
LIN {X 0,Y 453.561,Z 229.614,A -85,B 0,C 180,E1 -8448.379,E2 -8448.379} C_VEL
LIN {X 0,Y 453.579,Z 229.609,A -85,B 0,C 180,E1 -8451.086,E2 -8451.086} C_VEL
LIN {X 0,Y 453.644,Z 229.603,A -85,B 0,C 180,E1 -8453.774,E2 -8453.774} C_VEL
LIN {X 0,Y 453.746,Z 229.588,A -85,B 0,C 180,E1 -8457.337,E2 -8457.337} C_VEL
LIN {X 0,Y 453.819,Z 229.583,A -85,B 0,C 180,E1 -8460,E2 -8460} C_VEL
LIN {X 0,Y 453.734,Z 229.59,A -85,B 0,C 180,E1 -8462.663,E2 -8462.663} C_VEL
LIN {X 0,Y 453.671,Z 229.6,A -85,B 0,C 180,E1 -8466.225,E2 -8466.225} C_VEL
LIN {X 0,Y 453.593,Z 229.606,A -85,B 0,C 180,E1 -8468.913,E2 -8468.913} C_VEL
LIN {X 0,Y 453.566,Z 229.612,A -85,B 0,C 180,E1 -8472.529,E2 -8472.529} C_VEL
LIN {X 0,Y 453.547,Z 229.617,A -85,B 0,C 180,E1 -8476.196,E2 -8476.196} C_VEL
LIN {X 0,Y 453.522,Z 229.617,A -85,B 0,C 180,E1 -8479.041,E2 -8479.041} C_VEL
LIN {X 0,Y 453.478,Z 229.621,A -85,B 0,C 180,E1 -8481.836,E2 -8481.836} C_VEL
LIN {X 0,Y 453.503,Z 229.619,A -85,B 0,C 180,E1 -8484.735,E2 -8484.735} C_VEL
LIN {X 0,Y 453.533,Z 229.616,A -85,B 0,C 180,E1 -8487.959,E2 -8487.959} C_VEL
LIN {X 0,Y 453.466,Z 229.623,A -85,B 0,C 180,E1 -8491.525,E2 -8491.525} C_VEL
LIN {X 0,Y 453.484,Z 229.621,A -85,B 0,C 180,E1 -8494.776,E2 -8494.776} C_VEL
LIN {X 0,Y 453.459,Z 229.624,A -85,B 0,C 180,E1 -8498.312,E2 -8498.312} C_VEL
LIN {X 0,Y 453.471,Z 229.628,A -85,B 0,C 180,E1 -8500.612,E2 -8500.612} C_VEL
LIN {X 0,Y 453.461,Z 229.626,A -85,B 0,C 180,E1 -8504.222,E2 -8504.222} C_VEL
LIN {X 0,Y 453.465,Z 229.628,A -85,B 0,C 180,E1 -8507.005,E2 -8507.005} C_VEL
LIN {X 0,Y 453.472,Z 229.625,A -85,B 0,C 180,E1 -8509.413,E2 -8509.413} C_VEL
LIN {X 0,Y 453.458,Z 229.797,A -85,B 0,C 180,E1 -8510.547,E2 -8510.547} C_VEL
LIN {X 0,Y 453.516,Z 232.709,A -85,B 0,C 180,E1 -8512.816,E2 -8512.816} C_VEL
LIN {X 0,Y 453.489,Z 235.898,A -85,B 0,C 180,E1 -8515.223,E2 -8515.223} C_VEL
LIN {X 0,Y 453.274,Z 240.411,A -85,B 0,C 180,E1 -8518.515,E2 -8518.515} C_VEL
LIN {X 0,Y 453.089,Z 244.283,A -85,B 0,C 180,E1 -8521.259,E2 -8521.259} C_VEL
LIN {X 0,Y 452.972,Z 248.607,A -85,B 0,C 180,E1 -8524.251,E2 -8524.251} C_VEL
LIN {X 0,Y 452.875,Z 253.01,A -85,B 0,C 180,E1 -8527.172,E2 -8527.172} C_VEL
LIN {X 0,Y 452.773,Z 257.395,A -85,B 0,C 180,E1 -8530.033,E2 -8530.033} C_VEL
LIN {X 0,Y 452.767,Z 258.659,A -85,B 0,C 180,E1 -8530.829,E2 -8530.829} C_VEL
LIN {X 0,Y 456.485,Z 273.225,A -85,B 0,C 180,E1 -8531.362,E2 -8531.362} C_VEL
LIN {X 0,Y 458.3,Z 282.525,A -85,B 0,C 180,E1 -8531.776,E2 -8531.776} C_VEL
LIN {X 0,Y 457.721,Z 296.22,A -85,B 0,C 180,E1 -8532.412,E2 -8532.412} C_VEL
LIN {X 0,Y 457.036,Z 309.715,A -85,B 0,C 180,E1 -8533.242,E2 -8533.242} C_VEL
LIN {X 0,Y 456.212,Z 322.593,A -85,B 0,C 180,E1 -8534.246,E2 -8534.246} C_VEL
LIN {X 0,Y 455.498,Z 334.174,A -85,B 0,C 180,E1 -8535.365,E2 -8535.365} C_VEL
LIN {X 0,Y 455.014,Z 340.561,A -85,B 0,C 180,E1 -8536.084,E2 -8536.084} C_VEL
LIN {X 0,Y 454.054,Z 344.83,A -85,B 0,C 180,E1 -8536.586,E2 -8536.586} C_VEL
LIN {X 0,Y 450.842,Z 351.476,A -85,B 0,C 180,E1 -8537.424,E2 -8537.424} C_VEL
LIN {X 0,Y 447.627,Z 357.636,A -85,B 0,C 180,E1 -8538.33,E2 -8538.33} C_VEL
LIN {X 0,Y 446.672,Z 361.095,A -85,B 0,C 180,E1 -8538.932,E2 -8538.932} C_VEL
LIN {X 0,Y 446.2,Z 368.599,A -85,B 0,C 180,E1 -8540.481,E2 -8540.481} C_VEL
LIN {X 0,Y 445.885,Z 374.006,A -85,B 0,C 180,E1 -8541.845,E2 -8541.845} C_VEL
LIN {X 0,Y 445.666,Z 379.689,A -85,B 0,C 180,E1 -8543.662,E2 -8543.662} C_VEL
LIN {X 0,Y 445.435,Z 383.822,A -85,B 0,C 180,E1 -8545.475,E2 -8545.475} C_VEL
LIN {X 0,Y 445.437,Z 386.524,A -85,B 0,C 180,E1 -8547.287,E2 -8547.287} C_VEL
LIN {X 0,Y 445.313,Z 387.882,A -85,B 0,C 180,E1 -8549.096,E2 -8549.096} C_VEL
LIN {X 0,Y 445.314,Z 387.919,A -85,B 0,C 180,E1 -8550.904,E2 -8550.904} C_VEL
LIN {X 0,Y 445.437,Z 386.633,A -85,B 0,C 180,E1 -8552.713,E2 -8552.713} C_VEL
LIN {X 0,Y 445.433,Z 383.997,A -85,B 0,C 180,E1 -8554.525,E2 -8554.525} C_VEL
LIN {X 0,Y 445.647,Z 379.938,A -85,B 0,C 180,E1 -8556.338,E2 -8556.338} C_VEL
LIN {X 0,Y 445.867,Z 374.332,A -85,B 0,C 180,E1 -8558.156,E2 -8558.156} C_VEL
LIN {X 0,Y 446.239,Z 367.999,A -85,B 0,C 180,E1 -8559.748,E2 -8559.748} C_VEL
LIN {X 0,Y 446.749,Z 360.124,A -85,B 0,C 180,E1 -8561.341,E2 -8561.341} C_VEL
LIN {X 0,Y 447.331,Z 351.884,A -85,B 0,C 180,E1 -8562.706,E2 -8562.706} C_VEL
LIN {X 0,Y 448.02,Z 341.953,A -85,B 0,C 180,E1 -8564.072,E2 -8564.072} C_VEL
LIN {X 0,Y 448.848,Z 330.897,A -85,B 0,C 180,E1 -8565.321,E2 -8565.321} C_VEL
LIN {X 0,Y 449.621,Z 319.887,A -85,B 0,C 180,E1 -8566.341,E2 -8566.341} C_VEL
LIN {X 0,Y 450.354,Z 307.937,A -85,B 0,C 180,E1 -8567.248,E2 -8567.248} C_VEL
LIN {X 0,Y 451.026,Z 294.741,A -85,B 0,C 180,E1 -8568.041,E2 -8568.041} C_VEL
LIN {X 0,Y 451.522,Z 283.823,A -85,B 0,C 180,E1 -8568.551,E2 -8568.551} C_VEL
LIN {X 0,Y 449.863,Z 274.94,A -85,B 0,C 180,E1 -8568.966,E2 -8568.966} C_VEL
LIN {X 0,Y 446.097,Z 260.684,A -85,B 0,C 180,E1 -8569.526,E2 -8569.526} C_VEL
LIN {X 0,Y 445.708,Z 258.755,A -85,B 0,C 180,E1 -8569.589,E2 -8569.589} C_VEL
LIN {X 0,Y 445.779,Z 254.742,A -85,B 0,C 180,E1 -8572.233,E2 -8572.233} C_VEL
LIN {X 0,Y 445.884,Z 250.33,A -85,B 0,C 180,E1 -8575.187,E2 -8575.187} C_VEL
LIN {X 0,Y 446.008,Z 245.97,A -85,B 0,C 180,E1 -8578.212,E2 -8578.212} C_VEL
LIN {X 0,Y 446.209,Z 241.638,A -85,B 0,C 180,E1 -8581.317,E2 -8581.317} C_VEL
LIN {X 0,Y 446.411,Z 237.293,A -85,B 0,C 180,E1 -8584.525,E2 -8584.525} C_VEL
LIN {X 0,Y 446.463,Z 234.372,A -85,B 0,C 180,E1 -8586.74,E2 -8586.74} C_VEL
LIN {X 0,Y 446.418,Z 230.843,A -85,B 0,C 180,E1 -8589.519,E2 -8589.519} C_VEL
LIN {X 0,Y 446.41,Z 230.508,A -85,B 0,C 180,E1 -8590.915,E2 -8590.915} C_VEL
LIN {X 0,Y 446.404,Z 230.505,A -85,B 0,C 180,E1 -8593.846,E2 -8593.846} C_VEL
LIN {X 0,Y 446.397,Z 230.509,A -85,B 0,C 180,E1 -8596.404,E2 -8596.404} C_VEL
LIN {X 0,Y 446.405,Z 230.506,A -85,B 0,C 180,E1 -8599.798,E2 -8599.798} C_VEL
LIN {X 0,Y 446.409,Z 230.502,A -85,B 0,C 180,E1 -8602.121,E2 -8602.121} C_VEL
LIN {X 0,Y 446.426,Z 230.501,A -85,B 0,C 180,E1 -8605.477,E2 -8605.477} C_VEL
LIN {X 0,Y 446.417,Z 230.502,A -85,B 0,C 180,E1 -8608.7,E2 -8608.7} C_VEL
LIN {X 0,Y 446.488,Z 230.493,A -85,B 0,C 180,E1 -8611.821,E2 -8611.821} C_VEL
LIN {X 0,Y 446.447,Z 230.494,A -85,B 0,C 180,E1 -8614.847,E2 -8614.847} C_VEL
LIN {X 0,Y 446.451,Z 230.497,A -85,B 0,C 180,E1 -8618.245,E2 -8618.245} C_VEL
LIN {X 0,Y 446.454,Z 230.497,A -85,B 0,C 180,E1 -8621.649,E2 -8621.649} C_VEL
LIN {X 0,Y 446.511,Z 230.489,A -85,B 0,C 180,E1 -8624.48,E2 -8624.48} C_VEL
LIN {X 0,Y 446.52,Z 230.489,A -85,B 0,C 180,E1 -8628.193,E2 -8628.193} C_VEL
LIN {X 0,Y 446.535,Z 230.486,A -85,B 0,C 180,E1 -8630.944,E2 -8630.944} C_VEL
LIN {X 0,Y 446.639,Z 230.477,A -85,B 0,C 180,E1 -8633.676,E2 -8633.676} C_VEL
LIN {X 0,Y 446.683,Z 230.468,A -85,B 0,C 180,E1 -8637.294,E2 -8637.294} C_VEL
LIN {X 0,Y 446.764,Z 230.461,A -85,B 0,C 180,E1 -8640,E2 -8640} C_VEL
LIN {X 0,Y 446.694,Z 230.466,A -85,B 0,C 180,E1 -8642.705,E2 -8642.705} C_VEL
LIN {X 0,Y 446.614,Z 230.479,A -85,B 0,C 180,E1 -8646.324,E2 -8646.324} C_VEL
LIN {X 0,Y 446.529,Z 230.487,A -85,B 0,C 180,E1 -8649.055,E2 -8649.055} C_VEL
LIN {X 0,Y 446.525,Z 230.489,A -85,B 0,C 180,E1 -8652.73,E2 -8652.73} C_VEL
LIN {X 0,Y 446.498,Z 230.496,A -85,B 0,C 180,E1 -8656.227,E2 -8656.227} C_VEL
LIN {X 0,Y 446.471,Z 230.497,A -85,B 0,C 180,E1 -8659.303,E2 -8659.303} C_VEL
LIN {X 0,Y 446.421,Z 230.501,A -85,B 0,C 180,E1 -8662.199,E2 -8662.199} C_VEL
LIN {X 0,Y 446.44,Z 230.496,A -85,B 0,C 180,E1 -8665.153,E2 -8665.153} C_VEL
LIN {X 0,Y 446.438,Z 230.499,A -85,B 0,C 180,E1 -8668.182,E2 -8668.182} C_VEL
LIN {X 0,Y 446.417,Z 230.502,A -85,B 0,C 180,E1 -8671.3,E2 -8671.3} C_VEL
LIN {X 0,Y 446.431,Z 230.503,A -85,B 0,C 180,E1 -8674.523,E2 -8674.523} C_VEL
LIN {X 0,Y 446.415,Z 230.503,A -85,B 0,C 180,E1 -8678.079,E2 -8678.079} C_VEL
LIN {X 0,Y 446.429,Z 230.504,A -85,B 0,C 180,E1 -8680.917,E2 -8680.917} C_VEL
LIN {X 0,Y 446.402,Z 230.51,A -85,B 0,C 180,E1 -8683.846,E2 -8683.846} C_VEL
LIN {X 0,Y 446.431,Z 230.501,A -85,B 0,C 180,E1 -8686.779,E2 -8686.779} C_VEL
LIN {X 0,Y 446.487,Z 230.781,A -85,B 0,C 180,E1 -8687.402,E2 -8687.402} C_VEL
LIN {X 0,Y 447.16,Z 235.493,A -85,B 0,C 180,E1 -8690.366,E2 -8690.366} C_VEL
LIN {X 0,Y 447.289,Z 238.616,A -85,B 0,C 180,E1 -8692.209,E2 -8692.209} C_VEL
LIN {X 0,Y 446.979,Z 244.535,A -85,B 0,C 180,E1 -8695.525,E2 -8695.525} C_VEL
LIN {X 0,Y 446.728,Z 250.482,A -85,B 0,C 180,E1 -8698.724,E2 -8698.724} C_VEL
LIN {X 0,Y 446.521,Z 256.444,A -85,B 0,C 180,E1 -8701.824,E2 -8701.824} C_VEL
LIN {X 0,Y 446.132,Z 262.363,A -85,B 0,C 180,E1 -8704.828,E2 -8704.828} C_VEL
LIN {X 0,Y 445.947,Z 268.251,A -85,B 0,C 180,E1 -8707.776,E2 -8707.776} C_VEL
LIN {X 0,Y 445.758,Z 273.673,A -85,B 0,C 180,E1 -8710.437,E2 -8710.437} C_VEL
LIN {X 0,Y 449.249,Z 289.514,A -85,B 0,C 180,E1 -8711.002,E2 -8711.002} C_VEL
LIN {X 0,Y 451.26,Z 300.856,A -85,B 0,C 180,E1 -8711.518,E2 -8711.518} C_VEL
LIN {X 0,Y 450.673,Z 314.32,A -85,B 0,C 180,E1 -8712.178,E2 -8712.178} C_VEL
LIN {X 0,Y 449.859,Z 326.829,A -85,B 0,C 180,E1 -8712.967,E2 -8712.967} C_VEL
LIN {X 0,Y 449.008,Z 339.644,A -85,B 0,C 180,E1 -8713.986,E2 -8713.986} C_VEL
LIN {X 0,Y 448.222,Z 351.199,A -85,B 0,C 180,E1 -8715.122,E2 -8715.122} C_VEL
LIN {X 0,Y 447.521,Z 361.67,A -85,B 0,C 180,E1 -8716.375,E2 -8716.375} C_VEL
LIN {X 0,Y 446.891,Z 371.133,A -85,B 0,C 180,E1 -8717.742,E2 -8717.742} C_VEL
LIN {X 0,Y 446.375,Z 378.975,A -85,B 0,C 180,E1 -8719.109,E2 -8719.109} C_VEL
LIN {X 0,Y 445.988,Z 385.502,A -85,B 0,C 180,E1 -8720.476,E2 -8720.476} C_VEL
LIN {X 0,Y 445.704,Z 390.921,A -85,B 0,C 180,E1 -8721.841,E2 -8721.841} C_VEL
LIN {X 0,Y 445.529,Z 396.624,A -85,B 0,C 180,E1 -8723.66,E2 -8723.66} C_VEL
LIN {X 0,Y 445.394,Z 400.761,A -85,B 0,C 180,E1 -8725.475,E2 -8725.475} C_VEL
LIN {X 0,Y 445.394,Z 403.464,A -85,B 0,C 180,E1 -8727.287,E2 -8727.287} C_VEL
LIN {X 0,Y 445.312,Z 404.802,A -85,B 0,C 180,E1 -8729.096,E2 -8729.096} C_VEL
LIN {X 0,Y 445.312,Z 404.802,A -85,B 0,C 180,E1 -8730.904,E2 -8730.904} C_VEL
LIN {X 0,Y 445.394,Z 403.465,A -85,B 0,C 180,E1 -8732.713,E2 -8732.713} C_VEL
LIN {X 0,Y 445.394,Z 400.762,A -85,B 0,C 180,E1 -8734.525,E2 -8734.525} C_VEL
LIN {X 0,Y 445.509,Z 396.619,A -85,B 0,C 180,E1 -8736.34,E2 -8736.34} C_VEL
LIN {X 0,Y 445.704,Z 390.913,A -85,B 0,C 180,E1 -8738.159,E2 -8738.159} C_VEL
LIN {X 0,Y 446.07,Z 384.483,A -85,B 0,C 180,E1 -8739.751,E2 -8739.751} C_VEL
LIN {X 0,Y 446.541,Z 376.494,A -85,B 0,C 180,E1 -8741.346,E2 -8741.346} C_VEL
LIN {X 0,Y 447.094,Z 368.138,A -85,B 0,C 180,E1 -8742.713,E2 -8742.713} C_VEL
LIN {X 0,Y 447.759,Z 358.079,A -85,B 0,C 180,E1 -8744.081,E2 -8744.081} C_VEL
LIN {X 0,Y 448.531,Z 346.862,A -85,B 0,C 180,E1 -8745.332,E2 -8745.332} C_VEL
LIN {X 0,Y 449.266,Z 335.703,A -85,B 0,C 180,E1 -8746.354,E2 -8746.354} C_VEL
LIN {X 0,Y 450.093,Z 323.554,A -85,B 0,C 180,E1 -8747.258,E2 -8747.258} C_VEL
LIN {X 0,Y 450.835,Z 310.534,A -85,B 0,C 180,E1 -8748.025,E2 -8748.025} C_VEL
LIN {X 0,Y 451.253,Z 300.866,A -85,B 0,C 180,E1 -8748.478,E2 -8748.478} C_VEL
LIN {X 0,Y 448.759,Z 286.973,A -85,B 0,C 180,E1 -8749.098,E2 -8749.098} C_VEL
LIN {X 0,Y 445.764,Z 273.635,A -85,B 0,C 180,E1 -8749.577,E2 -8749.577} C_VEL
LIN {X 0,Y 445.945,Z 268.241,A -85,B 0,C 180,E1 -8752.224,E2 -8752.224} C_VEL
LIN {X 0,Y 446.129,Z 262.353,A -85,B 0,C 180,E1 -8755.172,E2 -8755.172} C_VEL
LIN {X 0,Y 446.523,Z 256.404,A -85,B 0,C 180,E1 -8758.188,E2 -8758.188} C_VEL
LIN {X 0,Y 446.756,Z 249.388,A -85,B 0,C 180,E1 -8761.844,E2 -8761.844} C_VEL
LIN {X 0,Y 446.98,Z 244.512,A -85,B 0,C 180,E1 -8764.474,E2 -8764.474} C_VEL
LIN {X 0,Y 447.219,Z 240.461,A -85,B 0,C 180,E1 -8766.73,E2 -8766.73} C_VEL
LIN {X 0,Y 447.244,Z 236.641,A -85,B 0,C 180,E1 -8768.944,E2 -8768.944} C_VEL
LIN {X 0,Y 446.795,Z 232.707,A -85,B 0,C 180,E1 -8771.35,E2 -8771.35} C_VEL
LIN {X 0,Y 446.44,Z 230.503,A -85,B 0,C 180,E1 -8772.834,E2 -8772.834} C_VEL
LIN {X 0,Y 446.452,Z 230.503,A -85,B 0,C 180,E1 -8775.104,E2 -8775.104} C_VEL
LIN {X 0,Y 446.429,Z 230.501,A -85,B 0,C 180,E1 -8778.609,E2 -8778.609} C_VEL
LIN {X 0,Y 446.442,Z 230.503,A -85,B 0,C 180,E1 -8780.973,E2 -8780.973} C_VEL
LIN {X 0,Y 446.418,Z 230.507,A -85,B 0,C 180,E1 -8784.374,E2 -8784.374} C_VEL
LIN {X 0,Y 446.423,Z 230.505,A -85,B 0,C 180,E1 -8787.639,E2 -8787.639} C_VEL
LIN {X 0,Y 446.427,Z 230.504,A -85,B 0,C 180,E1 -8790.789,E2 -8790.789} C_VEL
LIN {X 0,Y 446.437,Z 230.502,A -85,B 0,C 180,E1 -8793.846,E2 -8793.846} C_VEL
LIN {X 0,Y 446.426,Z 230.501,A -85,B 0,C 180,E1 -8796.823,E2 -8796.823} C_VEL
LIN {X 0,Y 446.444,Z 230.498,A -85,B 0,C 180,E1 -8799.737,E2 -8799.737} C_VEL
LIN {X 0,Y 446.453,Z 230.497,A -85,B 0,C 180,E1 -8802.597,E2 -8802.597} C_VEL
LIN {X 0,Y 446.474,Z 230.496,A -85,B 0,C 180,E1 -8805.413,E2 -8805.413} C_VEL
LIN {X 0,Y 446.519,Z 230.489,A -85,B 0,C 180,E1 -8808.193,E2 -8808.193} C_VEL
LIN {X 0,Y 446.528,Z 230.487,A -85,B 0,C 180,E1 -8810.944,E2 -8810.944} C_VEL
LIN {X 0,Y 446.613,Z 230.48,A -85,B 0,C 180,E1 -8813.676,E2 -8813.676} C_VEL
LIN {X 0,Y 446.693,Z 230.467,A -85,B 0,C 180,E1 -8817.295,E2 -8817.295} C_VEL
LIN {X 0,Y 446.789,Z 230.459,A -85,B 0,C 180,E1 -8820,E2 -8820} C_VEL
LIN {X 0,Y 446.682,Z 230.468,A -85,B 0,C 180,E1 -8822.706,E2 -8822.706} C_VEL
LIN {X 0,Y 446.641,Z 230.477,A -85,B 0,C 180,E1 -8826.324,E2 -8826.324} C_VEL
LIN {X 0,Y 446.539,Z 230.485,A -85,B 0,C 180,E1 -8829.055,E2 -8829.055} C_VEL
LIN {X 0,Y 446.523,Z 230.49,A -85,B 0,C 180,E1 -8832.73,E2 -8832.73} C_VEL
LIN {X 0,Y 446.492,Z 230.494,A -85,B 0,C 180,E1 -8836.459,E2 -8836.459} C_VEL
LIN {X 0,Y 446.471,Z 230.498,A -85,B 0,C 180,E1 -8839.303,E2 -8839.303} C_VEL
LIN {X 0,Y 446.42,Z 230.501,A -85,B 0,C 180,E1 -8842.2,E2 -8842.2} C_VEL
LIN {X 0,Y 446.446,Z 230.497,A -85,B 0,C 180,E1 -8845.153,E2 -8845.153} C_VEL
LIN {X 0,Y 446.487,Z 230.492,A -85,B 0,C 180,E1 -8848.179,E2 -8848.179} C_VEL
LIN {X 0,Y 446.42,Z 230.501,A -85,B 0,C 180,E1 -8851.775,E2 -8851.775} C_VEL
LIN {X 0,Y 446.425,Z 230.501,A -85,B 0,C 180,E1 -8854.524,E2 -8854.524} C_VEL
LIN {X 0,Y 446.413,Z 230.502,A -85,B 0,C 180,E1 -8858.079,E2 -8858.079} C_VEL
LIN {X 0,Y 446.408,Z 230.504,A -85,B 0,C 180,E1 -8861.394,E2 -8861.394} C_VEL
LIN {X 0,Y 446.452,Z 230.5,A -85,B 0,C 180,E1 -8865.104,E2 -8865.104} C_VEL
LIN {X 0,Y 446.421,Z 230.506,A -85,B 0,C 180,E1 -8868.608,E2 -8868.608} C_VEL
LIN {X 0,Y 446.428,Z 230.708,A -85,B 0,C 180,E1 -8870.48,E2 -8870.48} C_VEL
LIN {X 0,Y 446.473,Z 234.417,A -85,B 0,C 180,E1 -8873.399,E2 -8873.399} C_VEL
LIN {X 0,Y 446.41,Z 237.149,A -85,B 0,C 180,E1 -8875.475,E2 -8875.475} C_VEL
LIN {X 0,Y 446.209,Z 241.502,A -85,B 0,C 180,E1 -8878.683,E2 -8878.683} C_VEL
LIN {X 0,Y 445.997,Z 246.039,A -85,B 0,C 180,E1 -8881.939,E2 -8881.939} C_VEL
LIN {X 0,Y 445.883,Z 250.189,A -85,B 0,C 180,E1 -8884.813,E2 -8884.813} C_VEL
LIN {X 0,Y 445.779,Z 254.6,A -85,B 0,C 180,E1 -8887.767,E2 -8887.767} C_VEL
LIN {X 0,Y 445.717,Z 258.749,A -85,B 0,C 180,E1 -8890.501,E2 -8890.501} C_VEL
LIN {X 0,Y 449.75,Z 274.462,A -85,B 0,C 180,E1 -8891.108,E2 -8891.108} C_VEL
LIN {X 0,Y 451.409,Z 282.215,A -85,B 0,C 180,E1 -8891.469,E2 -8891.469} C_VEL
LIN {X 0,Y 451.019,Z 295.618,A -85,B 0,C 180,E1 -8892.099,E2 -8892.099} C_VEL
LIN {X 0,Y 450.325,Z 308.277,A -85,B 0,C 180,E1 -8892.868,E2 -8892.868} C_VEL
LIN {X 0,Y 449.582,Z 320.157,A -85,B 0,C 180,E1 -8893.774,E2 -8893.774} C_VEL
LIN {X 0,Y 448.747,Z 332.182,A -85,B 0,C 180,E1 -8894.908,E2 -8894.908} C_VEL
LIN {X 0,Y 447.935,Z 343.02,A -85,B 0,C 180,E1 -8896.157,E2 -8896.157} C_VEL
LIN {X 0,Y 447.283,Z 352.77,A -85,B 0,C 180,E1 -8897.523,E2 -8897.523} C_VEL
LIN {X 0,Y 446.672,Z 361.095,A -85,B 0,C 180,E1 -8898.932,E2 -8898.932} C_VEL
LIN {X 0,Y 445.721,Z 364.408,A -85,B 0,C 180,E1 -8899.55,E2 -8899.55} C_VEL
LIN {X 0,Y 442.548,Z 369.458,A -85,B 0,C 180,E1 -8900.574,E2 -8900.574} C_VEL
LIN {X 0,Y 439.485,Z 373.925,A -85,B 0,C 180,E1 -8901.654,E2 -8901.654} C_VEL
LIN {X 0,Y 438.715,Z 376.304,A -85,B 0,C 180,E1 -8902.353,E2 -8902.353} C_VEL
LIN {X 0,Y 438.572,Z 381.016,A -85,B 0,C 180,E1 -8904.021,E2 -8904.021} C_VEL
LIN {X 0,Y 438.363,Z 383.957,A -85,B 0,C 180,E1 -8905.402,E2 -8905.402} C_VEL
LIN {X 0,Y 438.365,Z 386.659,A -85,B 0,C 180,E1 -8907.243,E2 -8907.243} C_VEL
LIN {X 0,Y 438.228,Z 388.016,A -85,B 0,C 180,E1 -8909.081,E2 -8909.081} C_VEL
LIN {X 0,Y 438.229,Z 388.054,A -85,B 0,C 180,E1 -8910.919,E2 -8910.919} C_VEL
LIN {X 0,Y 438.365,Z 386.767,A -85,B 0,C 180,E1 -8912.757,E2 -8912.757} C_VEL
LIN {X 0,Y 438.361,Z 384.131,A -85,B 0,C 180,E1 -8914.598,E2 -8914.598} C_VEL
LIN {X 0,Y 438.594,Z 380.071,A -85,B 0,C 180,E1 -8916.44,E2 -8916.44} C_VEL
LIN {X 0,Y 438.83,Z 374.465,A -85,B 0,C 180,E1 -8918.287,E2 -8918.287} C_VEL
LIN {X 0,Y 439.217,Z 368.133,A -85,B 0,C 180,E1 -8919.905,E2 -8919.905} C_VEL
LIN {X 0,Y 439.782,Z 360.257,A -85,B 0,C 180,E1 -8921.523,E2 -8921.523} C_VEL
LIN {X 0,Y 440.353,Z 352.017,A -85,B 0,C 180,E1 -8922.911,E2 -8922.911} C_VEL
LIN {X 0,Y 441.111,Z 342.085,A -85,B 0,C 180,E1 -8924.297,E2 -8924.297} C_VEL
LIN {X 0,Y 441.995,Z 331.028,A -85,B 0,C 180,E1 -8925.565,E2 -8925.565} C_VEL
LIN {X 0,Y 442.806,Z 320.017,A -85,B 0,C 180,E1 -8926.6,E2 -8926.6} C_VEL
LIN {X 0,Y 443.685,Z 306.809,A -85,B 0,C 180,E1 -8927.601,E2 -8927.601} C_VEL
LIN {X 0,Y 444.322,Z 293.976,A -85,B 0,C 180,E1 -8928.37,E2 -8928.37} C_VEL
LIN {X 0,Y 444.703,Z 283.641,A -85,B 0,C 180,E1 -8928.86,E2 -8928.86} C_VEL
LIN {X 0,Y 441.542,Z 269.756,A -85,B 0,C 180,E1 -8929.512,E2 -8929.512} C_VEL
LIN {X 0,Y 438.668,Z 258.871,A -85,B 0,C 180,E1 -8929.927,E2 -8929.927} C_VEL
LIN {X 0,Y 438.794,Z 253.385,A -85,B 0,C 180,E1 -8933.604,E2 -8933.604} C_VEL
LIN {X 0,Y 438.875,Z 248.97,A -85,B 0,C 180,E1 -8936.64,E2 -8936.64} C_VEL
LIN {X 0,Y 439.114,Z 244.007,A -85,B 0,C 180,E1 -8940.2,E2 -8940.2} C_VEL
LIN {X 0,Y 439.303,Z 239.29,A -85,B 0,C 180,E1 -8943.705,E2 -8943.705} C_VEL
LIN {X 0,Y 439.421,Z 235.913,A -85,B 0,C 180,E1 -8946.283,E2 -8946.283} C_VEL
LIN {X 0,Y 439.433,Z 232.99,A -85,B 0,C 180,E1 -8948.59,E2 -8948.59} C_VEL
LIN {X 0,Y 439.347,Z 231.459,A -85,B 0,C 180,E1 -8949.84,E2 -8949.84} C_VEL
LIN {X 0,Y 439.384,Z 231.38,A -85,B 0,C 180,E1 -8952.627,E2 -8952.627} C_VEL
LIN {X 0,Y 439.403,Z 231.377,A -85,B 0,C 180,E1 -8955.271,E2 -8955.271} C_VEL
LIN {X 0,Y 439.359,Z 231.382,A -85,B 0,C 180,E1 -8959.017,E2 -8959.017} C_VEL
LIN {X 0,Y 439.37,Z 231.38,A -85,B 0,C 180,E1 -8961.609,E2 -8961.609} C_VEL
LIN {X 0,Y 439.399,Z 231.377,A -85,B 0,C 180,E1 -8964.844,E2 -8964.844} C_VEL
LIN {X 0,Y 439.374,Z 231.38,A -85,B 0,C 180,E1 -8968.139,E2 -8968.139} C_VEL
LIN {X 0,Y 439.435,Z 231.371,A -85,B 0,C 180,E1 -8971.598,E2 -8971.598} C_VEL
LIN {X 0,Y 439.401,Z 231.374,A -85,B 0,C 180,E1 -8974.415,E2 -8974.415} C_VEL
LIN {X 0,Y 439.367,Z 231.383,A -85,B 0,C 180,E1 -8977.425,E2 -8977.425} C_VEL
LIN {X 0,Y 439.444,Z 231.374,A -85,B 0,C 180,E1 -8980.663,E2 -8980.663} C_VEL
LIN {X 0,Y 439.465,Z 231.368,A -85,B 0,C 180,E1 -8984.225,E2 -8984.225} C_VEL
LIN {X 0,Y 439.486,Z 231.365,A -85,B 0,C 180,E1 -8988.001,E2 -8988.001} C_VEL
LIN {X 0,Y 439.507,Z 231.364,A -85,B 0,C 180,E1 -8991.725,E2 -8991.725} C_VEL
LIN {X 0,Y 439.618,Z 231.347,A -85,B 0,C 180,E1 -8994.496,E2 -8994.496} C_VEL
LIN {X 0,Y 439.635,Z 231.348,A -85,B 0,C 180,E1 -8998.168,E2 -8998.168} C_VEL
LIN {X 0,Y 439.713,Z 231.339,A -85,B 0,C 180,E1 -9000,E2 -9000} C_VEL
LIN {X 0,Y 439.643,Z 231.344,A -85,B 0,C 180,E1 -9002.749,E2 -9002.749} C_VEL
LIN {X 0,Y 439.566,Z 231.358,A -85,B 0,C 180,E1 -9006.426,E2 -9006.426} C_VEL
LIN {X 0,Y 439.493,Z 231.364,A -85,B 0,C 180,E1 -9009.202,E2 -9009.202} C_VEL
LIN {X 0,Y 439.469,Z 231.37,A -85,B 0,C 180,E1 -9012.937,E2 -9012.937} C_VEL
LIN {X 0,Y 439.448,Z 231.373,A -85,B 0,C 180,E1 -9016.348,E2 -9016.348} C_VEL
LIN {X 0,Y 439.404,Z 231.379,A -85,B 0,C 180,E1 -9019.626,E2 -9019.626} C_VEL
LIN {X 0,Y 439.366,Z 231.383,A -85,B 0,C 180,E1 -9022.575,E2 -9022.575} C_VEL
LIN {X 0,Y 439.377,Z 231.377,A -85,B 0,C 180,E1 -9025.587,E2 -9025.587} C_VEL
LIN {X 0,Y 439.391,Z 231.377,A -85,B 0,C 180,E1 -9028.675,E2 -9028.675} C_VEL
LIN {X 0,Y 439.372,Z 231.379,A -85,B 0,C 180,E1 -9032.03,E2 -9032.03} C_VEL
LIN {X 0,Y 439.395,Z 231.38,A -85,B 0,C 180,E1 -9035.34,E2 -9035.34} C_VEL
LIN {X 0,Y 439.378,Z 231.382,A -85,B 0,C 180,E1 -9038.595,E2 -9038.595} C_VEL
LIN {X 0,Y 439.39,Z 231.379,A -85,B 0,C 180,E1 -9041.257,E2 -9041.257} C_VEL
LIN {X 0,Y 439.401,Z 231.381,A -85,B 0,C 180,E1 -9044.729,E2 -9044.729} C_VEL
LIN {X 0,Y 439.392,Z 231.402,A -85,B 0,C 180,E1 -9046.991,E2 -9046.991} C_VEL
LIN {X 0,Y 440.1,Z 236.167,A -85,B 0,C 180,E1 -9050.042,E2 -9050.042} C_VEL
LIN {X 0,Y 440.275,Z 238.54,A -85,B 0,C 180,E1 -9051.497,E2 -9051.497} C_VEL
LIN {X 0,Y 440.052,Z 243.813,A -85,B 0,C 180,E1 -9054.539,E2 -9054.539} C_VEL
LIN {X 0,Y 439.761,Z 250.392,A -85,B 0,C 180,E1 -9058.171,E2 -9058.171} C_VEL
LIN {X 0,Y 439.473,Z 256.834,A -85,B 0,C 180,E1 -9061.589,E2 -9061.589} C_VEL
LIN {X 0,Y 439.115,Z 262.252,A -85,B 0,C 180,E1 -9064.397,E2 -9064.397} C_VEL
LIN {X 0,Y 438.906,Z 268.128,A -85,B 0,C 180,E1 -9067.399,E2 -9067.399} C_VEL
LIN {X 0,Y 438.718,Z 273.55,A -85,B 0,C 180,E1 -9070.115,E2 -9070.115} C_VEL
LIN {X 0,Y 442.195,Z 289.056,A -85,B 0,C 180,E1 -9070.676,E2 -9070.676} C_VEL
LIN {X 0,Y 444.464,Z 301.812,A -85,B 0,C 180,E1 -9071.275,E2 -9071.275} C_VEL
LIN {X 0,Y 443.838,Z 315.283,A -85,B 0,C 180,E1 -9071.96,E2 -9071.96} C_VEL
LIN {X 0,Y 442.956,Z 328.282,A -85,B 0,C 180,E1 -9072.812,E2 -9072.812} C_VEL
LIN {X 0,Y 442.062,Z 340.806,A -85,B 0,C 180,E1 -9073.846,E2 -9073.846} C_VEL
LIN {X 0,Y 441.246,Z 352.134,A -85,B 0,C 180,E1 -9075,E2 -9075} C_VEL
LIN {X 0,Y 440.45,Z 363.231,A -85,B 0,C 180,E1 -9076.387,E2 -9076.387} C_VEL
LIN {X 0,Y 439.83,Z 372.384,A -85,B 0,C 180,E1 -9077.777,E2 -9077.777} C_VEL
LIN {X 0,Y 439.183,Z 381.133,A -85,B 0,C 180,E1 -9079.395,E2 -9079.395} C_VEL
LIN {X 0,Y 438.826,Z 387.296,A -85,B 0,C 180,E1 -9080.784,E2 -9080.784} C_VEL
LIN {X 0,Y 438.511,Z 393.843,A -85,B 0,C 180,E1 -9082.633,E2 -9082.633} C_VEL
LIN {X 0,Y 438.374,Z 398.744,A -85,B 0,C 180,E1 -9084.48,E2 -9084.48} C_VEL
LIN {X 0,Y 438.248,Z 402.151,A -85,B 0,C 180,E1 -9086.322,E2 -9086.322} C_VEL
LIN {X 0,Y 438.271,Z 404.167,A -85,B 0,C 180,E1 -9088.162,E2 -9088.162} C_VEL
LIN {X 0,Y 438.226,Z 404.835,A -85,B 0,C 180,E1 -9090,E2 -9090} C_VEL
LIN {X 0,Y 438.271,Z 404.167,A -85,B 0,C 180,E1 -9091.838,E2 -9091.838} C_VEL
LIN {X 0,Y 438.248,Z 402.151,A -85,B 0,C 180,E1 -9093.678,E2 -9093.678} C_VEL
LIN {X 0,Y 438.371,Z 398.742,A -85,B 0,C 180,E1 -9095.52,E2 -9095.52} C_VEL
LIN {X 0,Y 438.511,Z 393.835,A -85,B 0,C 180,E1 -9097.366,E2 -9097.366} C_VEL
LIN {X 0,Y 438.826,Z 387.287,A -85,B 0,C 180,E1 -9099.216,E2 -9099.216} C_VEL
LIN {X 0,Y 439.253,Z 380.001,A -85,B 0,C 180,E1 -9100.836,E2 -9100.836} C_VEL
LIN {X 0,Y 439.816,Z 372.368,A -85,B 0,C 180,E1 -9102.224,E2 -9102.224} C_VEL
LIN {X 0,Y 440.431,Z 363.373,A -85,B 0,C 180,E1 -9103.59,E2 -9103.59} C_VEL
LIN {X 0,Y 441.099,Z 354.082,A -85,B 0,C 180,E1 -9104.769,E2 -9104.769} C_VEL
LIN {X 0,Y 441.898,Z 343.196,A -85,B 0,C 180,E1 -9105.923,E2 -9105.923} C_VEL
LIN {X 0,Y 442.764,Z 331.281,A -85,B 0,C 180,E1 -9106.958,E2 -9106.958} C_VEL
LIN {X 0,Y 443.614,Z 319.086,A -85,B 0,C 180,E1 -9107.81,E2 -9107.81} C_VEL
LIN {X 0,Y 444.27,Z 306.311,A -85,B 0,C 180,E1 -9108.516,E2 -9108.516} C_VEL
LIN {X 0,Y 444.456,Z 301.754,A -85,B 0,C 180,E1 -9108.723,E2 -9108.723} C_VEL
LIN {X 0,Y 441.89,Z 287.551,A -85,B 0,C 180,E1 -9109.383,E2 -9109.383} C_VEL
LIN {X 0,Y 438.712,Z 273.557,A -85,B 0,C 180,E1 -9109.878,E2 -9109.878} C_VEL
LIN {X 0,Y 438.902,Z 268.118,A -85,B 0,C 180,E1 -9112.601,E2 -9112.601} C_VEL
LIN {X 0,Y 439.114,Z 262.24,A -85,B 0,C 180,E1 -9115.603,E2 -9115.603} C_VEL
LIN {X 0,Y 439.477,Z 256.322,A -85,B 0,C 180,E1 -9118.669,E2 -9118.669} C_VEL
LIN {X 0,Y 439.748,Z 249.847,A -85,B 0,C 180,E1 -9122.109,E2 -9122.109} C_VEL
LIN {X 0,Y 440.063,Z 243.779,A -85,B 0,C 180,E1 -9125.463,E2 -9125.463} C_VEL
LIN {X 0,Y 440.235,Z 240.495,A -85,B 0,C 180,E1 -9127.347,E2 -9127.347} C_VEL
LIN {X 0,Y 440.166,Z 236.566,A -85,B 0,C 180,E1 -9129.693,E2 -9129.693} C_VEL
LIN {X 0,Y 439.504,Z 231.935,A -85,B 0,C 180,E1 -9132.644,E2 -9132.644} C_VEL
LIN {X 0,Y 439.404,Z 231.379,A -85,B 0,C 180,E1 -9133.118,E2 -9133.118} C_VEL
LIN {X 0,Y 439.366,Z 231.386,A -85,B 0,C 180,E1 -9136.039,E2 -9136.039} C_VEL
LIN {X 0,Y 439.381,Z 231.38,A -85,B 0,C 180,E1 -9139.019,E2 -9139.019} C_VEL
LIN {X 0,Y 439.373,Z 231.381,A -85,B 0,C 180,E1 -9141.608,E2 -9141.608} C_VEL
LIN {X 0,Y 439.399,Z 231.378,A -85,B 0,C 180,E1 -9144.844,E2 -9144.844} C_VEL
LIN {X 0,Y 439.374,Z 231.38,A -85,B 0,C 180,E1 -9148.14,E2 -9148.14} C_VEL
LIN {X 0,Y 439.402,Z 231.375,A -85,B 0,C 180,E1 -9151.606,E2 -9151.606} C_VEL
LIN {X 0,Y 439.377,Z 231.38,A -85,B 0,C 180,E1 -9154.413,E2 -9154.413} C_VEL
LIN {X 0,Y 439.365,Z 231.384,A -85,B 0,C 180,E1 -9157.425,E2 -9157.425} C_VEL
LIN {X 0,Y 439.442,Z 231.374,A -85,B 0,C 180,E1 -9160.663,E2 -9160.663} C_VEL
LIN {X 0,Y 439.464,Z 231.368,A -85,B 0,C 180,E1 -9164.225,E2 -9164.225} C_VEL
LIN {X 0,Y 439.485,Z 231.365,A -85,B 0,C 180,E1 -9168.001,E2 -9168.001} C_VEL
LIN {X 0,Y 439.503,Z 231.366,A -85,B 0,C 180,E1 -9171.725,E2 -9171.725} C_VEL
LIN {X 0,Y 439.606,Z 231.349,A -85,B 0,C 180,E1 -9174.496,E2 -9174.496} C_VEL
LIN {X 0,Y 439.636,Z 231.349,A -85,B 0,C 180,E1 -9178.168,E2 -9178.168} C_VEL
LIN {X 0,Y 439.758,Z 231.335,A -85,B 0,C 180,E1 -9180,E2 -9180} C_VEL
LIN {X 0,Y 439.631,Z 231.347,A -85,B 0,C 180,E1 -9182.749,E2 -9182.749} C_VEL
LIN {X 0,Y 439.613,Z 231.352,A -85,B 0,C 180,E1 -9186.425,E2 -9186.425} C_VEL
LIN {X 0,Y 439.501,Z 231.363,A -85,B 0,C 180,E1 -9189.202,E2 -9189.202} C_VEL
LIN {X 0,Y 439.467,Z 231.371,A -85,B 0,C 180,E1 -9192.938,E2 -9192.938} C_VEL
LIN {X 0,Y 439.45,Z 231.373,A -85,B 0,C 180,E1 -9196.349,E2 -9196.349} C_VEL
LIN {X 0,Y 439.405,Z 231.377,A -85,B 0,C 180,E1 -9199.626,E2 -9199.626} C_VEL
LIN {X 0,Y 439.366,Z 231.382,A -85,B 0,C 180,E1 -9202.576,E2 -9202.576} C_VEL
LIN {X 0,Y 439.4,Z 231.377,A -85,B 0,C 180,E1 -9205.585,E2 -9205.585} C_VEL
LIN {X 0,Y 439.419,Z 231.373,A -85,B 0,C 180,E1 -9208.674,E2 -9208.674} C_VEL
LIN {X 0,Y 439.37,Z 231.38,A -85,B 0,C 180,E1 -9212.03,E2 -9212.03} C_VEL
LIN {X 0,Y 439.394,Z 231.378,A -85,B 0,C 180,E1 -9215.34,E2 -9215.34} C_VEL
LIN {X 0,Y 439.369,Z 231.381,A -85,B 0,C 180,E1 -9218.597,E2 -9218.597} C_VEL
LIN {X 0,Y 439.368,Z 231.381,A -85,B 0,C 180,E1 -9221.254,E2 -9221.254} C_VEL
LIN {X 0,Y 439.4,Z 231.377,A -85,B 0,C 180,E1 -9224.73,E2 -9224.73} C_VEL
LIN {X 0,Y 439.396,Z 231.379,A -85,B 0,C 180,E1 -9227.796,E2 -9227.796} C_VEL
LIN {X 0,Y 439.359,Z 231.393,A -85,B 0,C 180,E1 -9230.22,E2 -9230.22} C_VEL
LIN {X 0,Y 439.439,Z 234.319,A -85,B 0,C 180,E1 -9232.574,E2 -9232.574} C_VEL
LIN {X 0,Y 439.418,Z 237.235,A -85,B 0,C 180,E1 -9234.846,E2 -9234.846} C_VEL
LIN {X 0,Y 439.19,Z 241.595,A -85,B 0,C 180,E1 -9238.125,E2 -9238.125} C_VEL
LIN {X 0,Y 438.979,Z 245.931,A -85,B 0,C 180,E1 -9241.295,E2 -9241.295} C_VEL
LIN {X 0,Y 438.84,Z 250.308,A -85,B 0,C 180,E1 -9244.38,E2 -9244.38} C_VEL
LIN {X 0,Y 438.794,Z 253.244,A -85,B 0,C 180,E1 -9246.396,E2 -9246.396} C_VEL
LIN {X 0,Y 438.661,Z 258.398,A -85,B 0,C 180,E1 -9249.852,E2 -9249.852} C_VEL
LIN {X 0,Y 438.661,Z 259.059,A -85,B 0,C 180,E1 -9250.188,E2 -9250.188} C_VEL
LIN {X 0,Y 442.632,Z 274.058,A -85,B 0,C 180,E1 -9250.774,E2 -9250.774} C_VEL
LIN {X 0,Y 444.694,Z 284.283,A -85,B 0,C 180,E1 -9251.263,E2 -9251.263} C_VEL
LIN {X 0,Y 444.132,Z 297.635,A -85,B 0,C 180,E1 -9251.924,E2 -9251.924} C_VEL
LIN {X 0,Y 443.46,Z 309.997,A -85,B 0,C 180,E1 -9252.713,E2 -9252.713} C_VEL
LIN {X 0,Y 442.546,Z 322.873,A -85,B 0,C 180,E1 -9253.746,E2 -9253.746} C_VEL
LIN {X 0,Y 441.737,Z 334.453,A -85,B 0,C 180,E1 -9254.899,E2 -9254.899} C_VEL
LIN {X 0,Y 440.9,Z 344.934,A -85,B 0,C 180,E1 -9256.167,E2 -9256.167} C_VEL
LIN {X 0,Y 440.314,Z 352.909,A -85,B 0,C 180,E1 -9257.322,E2 -9257.322} C_VEL
LIN {X 0,Y 439.63,Z 361.638,A -85,B 0,C 180,E1 -9258.829,E2 -9258.829} C_VEL
LIN {X 0,Y 439.188,Z 368.736,A -85,B 0,C 180,E1 -9260.327,E2 -9260.327} C_VEL
LIN {X 0,Y 438.849,Z 374.143,A -85,B 0,C 180,E1 -9261.713,E2 -9261.713} C_VEL
LIN {X 0,Y 438.715,Z 376.304,A -85,B 0,C 180,E1 -9262.353,E2 -9262.353} C_VEL
LIN {X 0,Y 437.943,Z 378.54,A -85,B 0,C 180,E1 -9263.065,E2 -9263.065} C_VEL
LIN {X 0,Y 434.913,Z 381.687,A -85,B 0,C 180,E1 -9264.235,E2 -9264.235} C_VEL
LIN {X 0,Y 432.397,Z 383.797,A -85,B 0,C 180,E1 -9265.194,E2 -9265.194} C_VEL
LIN {X 0,Y 431.318,Z 385.127,A -85,B 0,C 180,E1 -9265.946,E2 -9265.946} C_VEL
LIN {X 0,Y 431.229,Z 385.519,A -85,B 0,C 180,E1 -9266.202,E2 -9266.202} C_VEL
LIN {X 0,Y 431.276,Z 386.794,A -85,B 0,C 180,E1 -9267.198,E2 -9267.198} C_VEL
LIN {X 0,Y 431.147,Z 388.151,A -85,B 0,C 180,E1 -9269.066,E2 -9269.066} C_VEL
LIN {X 0,Y 431.147,Z 388.188,A -85,B 0,C 180,E1 -9270.934,E2 -9270.934} C_VEL
LIN {X 0,Y 431.276,Z 386.901,A -85,B 0,C 180,E1 -9272.802,E2 -9272.802} C_VEL
LIN {X 0,Y 431.291,Z 384.264,A -85,B 0,C 180,E1 -9274.674,E2 -9274.674} C_VEL
LIN {X 0,Y 431.523,Z 380.205,A -85,B 0,C 180,E1 -9276.546,E2 -9276.546} C_VEL
LIN {X 0,Y 431.78,Z 374.599,A -85,B 0,C 180,E1 -9278.424,E2 -9278.424} C_VEL
LIN {X 0,Y 432.2,Z 368.266,A -85,B 0,C 180,E1 -9280.067,E2 -9280.067} C_VEL
LIN {X 0,Y 432.819,Z 360.389,A -85,B 0,C 180,E1 -9281.711,E2 -9281.711} C_VEL
LIN {X 0,Y 433.342,Z 352.15,A -85,B 0,C 180,E1 -9283.124,E2 -9283.124} C_VEL
LIN {X 0,Y 434.233,Z 342.217,A -85,B 0,C 180,E1 -9284.529,E2 -9284.529} C_VEL
LIN {X 0,Y 435.131,Z 331.159,A -85,B 0,C 180,E1 -9285.817,E2 -9285.817} C_VEL
LIN {X 0,Y 435.992,Z 320.147,A -85,B 0,C 180,E1 -9286.867,E2 -9286.867} C_VEL
LIN {X 0,Y 436.924,Z 307.041,A -85,B 0,C 180,E1 -9287.876,E2 -9287.876} C_VEL
LIN {X 0,Y 437.601,Z 293.897,A -85,B 0,C 180,E1 -9288.673,E2 -9288.673} C_VEL
LIN {X 0,Y 437.962,Z 284.917,A -85,B 0,C 180,E1 -9289.108,E2 -9289.108} C_VEL
LIN {X 0,Y 434.985,Z 271.729,A -85,B 0,C 180,E1 -9289.757,E2 -9289.757} C_VEL
LIN {X 0,Y 431.596,Z 259.003,A -85,B 0,C 180,E1 -9290.268,E2 -9290.268} C_VEL
LIN {X 0,Y 431.777,Z 253.514,A -85,B 0,C 180,E1 -9294.012,E2 -9294.012} C_VEL
LIN {X 0,Y 431.827,Z 249.081,A -85,B 0,C 180,E1 -9297.11,E2 -9297.11} C_VEL
LIN {X 0,Y 432.064,Z 244.51,A -85,B 0,C 180,E1 -9300.446,E2 -9300.446} C_VEL
LIN {X 0,Y 432.287,Z 239.824,A -85,B 0,C 180,E1 -9303.989,E2 -9303.989} C_VEL
LIN {X 0,Y 432.382,Z 235.996,A -85,B 0,C 180,E1 -9306.971,E2 -9306.971} C_VEL
LIN {X 0,Y 432.348,Z 233.065,A -85,B 0,C 180,E1 -9309.343,E2 -9309.343} C_VEL
LIN {X 0,Y 432.292,Z 232.268,A -85,B 0,C 180,E1 -9310.172,E2 -9310.172} C_VEL
LIN {X 0,Y 432.32,Z 232.262,A -85,B 0,C 180,E1 -9313.061,E2 -9313.061} C_VEL
LIN {X 0,Y 432.335,Z 232.257,A -85,B 0,C 180,E1 -9315.665,E2 -9315.665} C_VEL
LIN {X 0,Y 432.314,Z 232.26,A -85,B 0,C 180,E1 -9318.401,E2 -9318.401} C_VEL
LIN {X 0,Y 432.334,Z 232.256,A -85,B 0,C 180,E1 -9321.85,E2 -9321.85} C_VEL
LIN {X 0,Y 432.34,Z 232.255,A -85,B 0,C 180,E1 -9325.323,E2 -9325.323} C_VEL
LIN {X 0,Y 432.323,Z 232.257,A -85,B 0,C 180,E1 -9328.654,E2 -9328.654} C_VEL
LIN {X 0,Y 432.384,Z 232.25,A -85,B 0,C 180,E1 -9331.877,E2 -9331.877} C_VEL
LIN {X 0,Y 432.349,Z 232.25,A -85,B 0,C 180,E1 -9334.999,E2 -9334.999} C_VEL
LIN {X 0,Y 432.361,Z 232.252,A -85,B 0,C 180,E1 -9338.046,E2 -9338.046} C_VEL
LIN {X 0,Y 432.387,Z 232.25,A -85,B 0,C 180,E1 -9341.03,E2 -9341.03} C_VEL
LIN {X 0,Y 432.433,Z 232.246,A -85,B 0,C 180,E1 -9343.961,E2 -9343.961} C_VEL
LIN {X 0,Y 432.462,Z 232.24,A -85,B 0,C 180,E1 -9347.803,E2 -9347.803} C_VEL
LIN {X 0,Y 432.467,Z 232.24,A -85,B 0,C 180,E1 -9351.59,E2 -9351.59} C_VEL
LIN {X 0,Y 432.595,Z 232.222,A -85,B 0,C 180,E1 -9354.406,E2 -9354.406} C_VEL
LIN {X 0,Y 432.604,Z 232.223,A -85,B 0,C 180,E1 -9358.138,E2 -9358.138} C_VEL
LIN {X 0,Y 432.573,Z 232.226,A -85,B 0,C 180,E1 -9360.931,E2 -9360.931} C_VEL
LIN {X 0,Y 432.595,Z 232.222,A -85,B 0,C 180,E1 -9362.794,E2 -9362.794} C_VEL
LIN {X 0,Y 432.581,Z 232.225,A -85,B 0,C 180,E1 -9365.594,E2 -9365.594} C_VEL
LIN {X 0,Y 432.465,Z 232.242,A -85,B 0,C 180,E1 -9368.41,E2 -9368.41} C_VEL
LIN {X 0,Y 432.462,Z 232.239,A -85,B 0,C 180,E1 -9372.196,E2 -9372.196} C_VEL
LIN {X 0,Y 432.433,Z 232.247,A -85,B 0,C 180,E1 -9376.039,E2 -9376.039} C_VEL
LIN {X 0,Y 432.389,Z 232.253,A -85,B 0,C 180,E1 -9379.485,E2 -9379.485} C_VEL
LIN {X 0,Y 432.319,Z 232.26,A -85,B 0,C 180,E1 -9382.964,E2 -9382.964} C_VEL
LIN {X 0,Y 432.339,Z 232.253,A -85,B 0,C 180,E1 -9385.002,E2 -9385.002} C_VEL
LIN {X 0,Y 432.348,Z 232.254,A -85,B 0,C 180,E1 -9388.622,E2 -9388.622} C_VEL
LIN {X 0,Y 432.322,Z 232.257,A -85,B 0,C 180,E1 -9391.346,E2 -9391.346} C_VEL
LIN {X 0,Y 432.341,Z 232.257,A -85,B 0,C 180,E1 -9394.677,E2 -9394.677} C_VEL
LIN {X 0,Y 432.337,Z 232.257,A -85,B 0,C 180,E1 -9398.15,E2 -9398.15} C_VEL
LIN {X 0,Y 432.334,Z 232.258,A -85,B 0,C 180,E1 -9401.602,E2 -9401.602} C_VEL
LIN {X 0,Y 432.335,Z 232.262,A -85,B 0,C 180,E1 -9404.347,E2 -9404.347} C_VEL
LIN {X 0,Y 432.377,Z 232.353,A -85,B 0,C 180,E1 -9406.787,E2 -9406.787} C_VEL
LIN {X 0,Y 433.022,Z 236.832,A -85,B 0,C 180,E1 -9409.713,E2 -9409.713} C_VEL
LIN {X 0,Y 433.226,Z 240.44,A -85,B 0,C 180,E1 -9411.942,E2 -9411.942} C_VEL
LIN {X 0,Y 433.042,Z 244.372,A -85,B 0,C 180,E1 -9414.249,E2 -9414.249} C_VEL
LIN {X 0,Y 432.74,Z 250.351,A -85,B 0,C 180,E1 -9417.62,E2 -9417.62} C_VEL
LIN {X 0,Y 432.441,Z 256.238,A -85,B 0,C 180,E1 -9420.82,E2 -9420.82} C_VEL
LIN {X 0,Y 432.132,Z 262.142,A -85,B 0,C 180,E1 -9423.952,E2 -9423.952} C_VEL
LIN {X 0,Y 431.845,Z 268.006,A -85,B 0,C 180,E1 -9427.009,E2 -9427.009} C_VEL
LIN {X 0,Y 431.67,Z 273.562,A -85,B 0,C 180,E1 -9429.782,E2 -9429.782} C_VEL
LIN {X 0,Y 435.019,Z 288.059,A -85,B 0,C 180,E1 -9430.316,E2 -9430.316} C_VEL
LIN {X 0,Y 437.383,Z 301.073,A -85,B 0,C 180,E1 -9430.932,E2 -9430.932} C_VEL
LIN {X 0,Y 437.626,Z 305.201,A -85,B 0,C 180,E1 -9431.136,E2 -9431.136} C_VEL
LIN {X 0,Y 436.905,Z 317.878,A -85,B 0,C 180,E1 -9431.831,E2 -9431.831} C_VEL
LIN {X 0,Y 435.949,Z 331.185,A -85,B 0,C 180,E1 -9432.769,E2 -9432.769} C_VEL
LIN {X 0,Y 435.046,Z 343.094,A -85,B 0,C 180,E1 -9433.819,E2 -9433.819} C_VEL
LIN {X 0,Y 434.19,Z 353.974,A -85,B 0,C 180,E1 -9434.99,E2 -9434.99} C_VEL
LIN {X 0,Y 433.369,Z 364.731,A -85,B 0,C 180,E1 -9436.4,E2 -9436.4} C_VEL
LIN {X 0,Y 432.73,Z 373.609,A -85,B 0,C 180,E1 -9437.811,E2 -9437.811} C_VEL
LIN {X 0,Y 432.086,Z 382.119,A -85,B 0,C 180,E1 -9439.456,E2 -9439.456} C_VEL
LIN {X 0,Y 431.674,Z 388.979,A -85,B 0,C 180,E1 -9441.102,E2 -9441.102} C_VEL
LIN {X 0,Y 431.423,Z 393.708,A -85,B 0,C 180,E1 -9442.512,E2 -9442.512} C_VEL
LIN {X 0,Y 431.354,Z 396.886,A -85,B 0,C 180,E1 -9443.651,E2 -9443.651} C_VEL
LIN {X 0,Y 431.245,Z 400.492,A -85,B 0,C 180,E1 -9445.326,E2 -9445.326} C_VEL
LIN {X 0,Y 431.185,Z 403.195,A -85,B 0,C 180,E1 -9447.197,E2 -9447.197} C_VEL
LIN {X 0,Y 431.145,Z 404.533,A -85,B 0,C 180,E1 -9449.066,E2 -9449.066} C_VEL
LIN {X 0,Y 431.145,Z 404.533,A -85,B 0,C 180,E1 -9450.934,E2 -9450.934} C_VEL
LIN {X 0,Y 431.185,Z 403.195,A -85,B 0,C 180,E1 -9452.803,E2 -9452.803} C_VEL
LIN {X 0,Y 431.244,Z 400.492,A -85,B 0,C 180,E1 -9454.674,E2 -9454.674} C_VEL
LIN {X 0,Y 431.374,Z 396.348,A -85,B 0,C 180,E1 -9456.548,E2 -9456.548} C_VEL
LIN {X 0,Y 431.589,Z 390.641,A -85,B 0,C 180,E1 -9458.427,E2 -9458.427} C_VEL
LIN {X 0,Y 431.953,Z 384.208,A -85,B 0,C 180,E1 -9460.073,E2 -9460.073} C_VEL
LIN {X 0,Y 432.544,Z 376.22,A -85,B 0,C 180,E1 -9461.718,E2 -9461.718} C_VEL
LIN {X 0,Y 433.169,Z 367.259,A -85,B 0,C 180,E1 -9463.226,E2 -9463.226} C_VEL
LIN {X 0,Y 433.88,Z 357.803,A -85,B 0,C 180,E1 -9464.541,E2 -9464.541} C_VEL
LIN {X 0,Y 434.757,Z 346.585,A -85,B 0,C 180,E1 -9465.83,E2 -9465.83} C_VEL
LIN {X 0,Y 435.618,Z 335.426,A -85,B 0,C 180,E1 -9466.882,E2 -9466.882} C_VEL
LIN {X 0,Y 436.541,Z 323.276,A -85,B 0,C 180,E1 -9467.811,E2 -9467.811} C_VEL
LIN {X 0,Y 437.328,Z 309.838,A -85,B 0,C 180,E1 -9468.624,E2 -9468.624} C_VEL
LIN {X 0,Y 437.629,Z 302.444,A -85,B 0,C 180,E1 -9468.988,E2 -9468.988} C_VEL
LIN {X 0,Y 435.006,Z 288.061,A -85,B 0,C 180,E1 -9469.68,E2 -9469.68} C_VEL
LIN {X 0,Y 431.633,Z 273.424,A -85,B 0,C 180,E1 -9470.218,E2 -9470.218} C_VEL
LIN {X 0,Y 431.841,Z 267.995,A -85,B 0,C 180,E1 -9472.991,E2 -9472.991} C_VEL
LIN {X 0,Y 432.225,Z 261.111,A -85,B 0,C 180,E1 -9476.581,E2 -9476.581} C_VEL
LIN {X 0,Y 432.435,Z 256.217,A -85,B 0,C 180,E1 -9479.181,E2 -9479.181} C_VEL
LIN {X 0,Y 432.736,Z 250.26,A -85,B 0,C 180,E1 -9482.408,E2 -9482.408} C_VEL
LIN {X 0,Y 433.059,Z 244.324,A -85,B 0,C 180,E1 -9485.763,E2 -9485.763} C_VEL
LIN {X 0,Y 433.228,Z 240.418,A -85,B 0,C 180,E1 -9488.058,E2 -9488.058} C_VEL
LIN {X 0,Y 432.981,Z 236.494,A -85,B 0,C 180,E1 -9490.486,E2 -9490.486} C_VEL
LIN {X 0,Y 432.347,Z 232.259,A -85,B 0,C 180,E1 -9493.377,E2 -9493.377} C_VEL
LIN {X 0,Y 432.318,Z 232.261,A -85,B 0,C 180,E1 -9496.939,E2 -9496.939} C_VEL
LIN {X 0,Y 432.334,Z 232.259,A -85,B 0,C 180,E1 -9499.821,E2 -9499.821} C_VEL
LIN {X 0,Y 432.306,Z 232.263,A -85,B 0,C 180,E1 -9503.022,E2 -9503.022} C_VEL
LIN {X 0,Y 432.36,Z 232.258,A -85,B 0,C 180,E1 -9505.997,E2 -9505.997} C_VEL
LIN {X 0,Y 432.347,Z 232.256,A -85,B 0,C 180,E1 -9509.49,E2 -9509.49} C_VEL
LIN {X 0,Y 432.343,Z 232.255,A -85,B 0,C 180,E1 -9511.874,E2 -9511.874} C_VEL
LIN {X 0,Y 432.378,Z 232.254,A -85,B 0,C 180,E1 -9515.539,E2 -9515.539} C_VEL
LIN {X 0,Y 432.351,Z 232.257,A -85,B 0,C 180,E1 -9519.046,E2 -9519.046} C_VEL
LIN {X 0,Y 432.359,Z 232.255,A -85,B 0,C 180,E1 -9522.01,E2 -9522.01} C_VEL
LIN {X 0,Y 432.398,Z 232.248,A -85,B 0,C 180,E1 -9524.927,E2 -9524.927} C_VEL
LIN {X 0,Y 432.461,Z 232.24,A -85,B 0,C 180,E1 -9527.804,E2 -9527.804} C_VEL
LIN {X 0,Y 432.463,Z 232.241,A -85,B 0,C 180,E1 -9531.59,E2 -9531.59} C_VEL
LIN {X 0,Y 432.579,Z 232.225,A -85,B 0,C 180,E1 -9534.406,E2 -9534.406} C_VEL
LIN {X 0,Y 432.605,Z 232.224,A -85,B 0,C 180,E1 -9538.138,E2 -9538.138} C_VEL
LIN {X 0,Y 432.727,Z 232.21,A -85,B 0,C 180,E1 -9540,E2 -9540} C_VEL
LIN {X 0,Y 432.583,Z 232.225,A -85,B 0,C 180,E1 -9542.794,E2 -9542.794} C_VEL
LIN {X 0,Y 432.567,Z 232.23,A -85,B 0,C 180,E1 -9546.53,E2 -9546.53} C_VEL
LIN {X 0,Y 432.443,Z 232.243,A -85,B 0,C 180,E1 -9549.353,E2 -9549.353} C_VEL
LIN {X 0,Y 432.433,Z 232.246,A -85,B 0,C 180,E1 -9552.803,E2 -9552.803} C_VEL
LIN {X 0,Y 432.415,Z 232.248,A -85,B 0,C 180,E1 -9556.479,E2 -9556.479} C_VEL
LIN {X 0,Y 432.341,Z 232.254,A -85,B 0,C 180,E1 -9559.96,E2 -9559.96} C_VEL
LIN {X 0,Y 432.319,Z 232.259,A -85,B 0,C 180,E1 -9562.964,E2 -9562.964} C_VEL
LIN {X 0,Y 432.363,Z 232.255,A -85,B 0,C 180,E1 -9566.033,E2 -9566.033} C_VEL
LIN {X 0,Y 432.344,Z 232.258,A -85,B 0,C 180,E1 -9569.188,E2 -9569.188} C_VEL
LIN {X 0,Y 432.324,Z 232.26,A -85,B 0,C 180,E1 -9572.443,E2 -9572.443} C_VEL
LIN {X 0,Y 432.344,Z 232.258,A -85,B 0,C 180,E1 -9575.632,E2 -9575.632} C_VEL
LIN {X 0,Y 432.331,Z 232.259,A -85,B 0,C 180,E1 -9578.713,E2 -9578.713} C_VEL
LIN {X 0,Y 432.31,Z 232.262,A -85,B 0,C 180,E1 -9581.8,E2 -9581.8} C_VEL
LIN {X 0,Y 432.335,Z 232.257,A -85,B 0,C 180,E1 -9584.347,E2 -9584.347} C_VEL
LIN {X 0,Y 432.321,Z 232.262,A -85,B 0,C 180,E1 -9587.016,E2 -9587.016} C_VEL
LIN {X 0,Y 432.311,Z 232.262,A -85,B 0,C 180,E1 -9589.825,E2 -9589.825} C_VEL
LIN {X 0,Y 432.396,Z 233.685,A -85,B 0,C 180,E1 -9591.277,E2 -9591.277} C_VEL
LIN {X 0,Y 432.389,Z 237.544,A -85,B 0,C 180,E1 -9594.36,E2 -9594.36} C_VEL
LIN {X 0,Y 432.163,Z 241.948,A -85,B 0,C 180,E1 -9597.741,E2 -9597.741} C_VEL
LIN {X 0,Y 431.947,Z 246.036,A -85,B 0,C 180,E1 -9600.783,E2 -9600.783} C_VEL
LIN {X 0,Y 431.805,Z 250.422,A -85,B 0,C 180,E1 -9603.931,E2 -9603.931} C_VEL
LIN {X 0,Y 431.672,Z 254.847,A -85,B 0,C 180,E1 -9606.999,E2 -9606.999} C_VEL
LIN {X 0,Y 431.598,Z 259.143,A -85,B 0,C 180,E1 -9609.849,E2 -9609.849} C_VEL
LIN {X 0,Y 435.502,Z 273.826,A -85,B 0,C 180,E1 -9610.433,E2 -9610.433} C_VEL
LIN {X 0,Y 437.949,Z 285.566,A -85,B 0,C 180,E1 -9611.017,E2 -9611.017} C_VEL
LIN {X 0,Y 437.35,Z 298.56,A -85,B 0,C 180,E1 -9611.681,E2 -9611.681} C_VEL
LIN {X 0,Y 436.593,Z 311.716,A -85,B 0,C 180,E1 -9612.554,E2 -9612.554} C_VEL
LIN {X 0,Y 435.641,Z 324.3,A -85,B 0,C 180,E1 -9613.601,E2 -9613.601} C_VEL
LIN {X 0,Y 434.803,Z 335.658,A -85,B 0,C 180,E1 -9614.772,E2 -9614.772} C_VEL
LIN {X 0,Y 433.895,Z 346.201,A -85,B 0,C 180,E1 -9616.092,E2 -9616.092} C_VEL
LIN {X 0,Y 433.267,Z 354.526,A -85,B 0,C 180,E1 -9617.351,E2 -9617.351} C_VEL
LIN {X 0,Y 432.501,Z 363.545,A -85,B 0,C 180,E1 -9618.993,E2 -9618.993} C_VEL
LIN {X 0,Y 432.017,Z 370.805,A -85,B 0,C 180,E1 -9620.638,E2 -9620.638} C_VEL
LIN {X 0,Y 431.619,Z 377.324,A -85,B 0,C 180,E1 -9622.515,E2 -9622.515} C_VEL
LIN {X 0,Y 431.442,Z 382.211,A -85,B 0,C 180,E1 -9624.391,E2 -9624.391} C_VEL
LIN {X 0,Y 431.229,Z 385.519,A -85,B 0,C 180,E1 -9626.202,E2 -9626.202} C_VEL
LIN {X 0,Y 430.547,Z 386.635,A -85,B 0,C 180,E1 -9626.968,E2 -9626.968} C_VEL
LIN {X 0,Y 427.644,Z 387.887,A -85,B 0,C 180,E1 -9628.223,E2 -9628.223} C_VEL
LIN {X 0,Y 425.191,Z 388.371,A -85,B 0,C 180,E1 -9629.243,E2 -9629.243} C_VEL
LIN {X 0,Y 424.137,Z 388.47,A -85,B 0,C 180,E1 -9630.033,E2 -9630.033} C_VEL
LIN {X 0,Y 424.05,Z 388.422,A -85,B 0,C 180,E1 -9630.301,E2 -9630.301} C_VEL
LIN {X 0,Y 424.129,Z 387.845,A -85,B 0,C 180,E1 -9631.899,E2 -9631.899} C_VEL
LIN {X 0,Y 424.135,Z 385.89,A -85,B 0,C 180,E1 -9633.801,E2 -9633.801} C_VEL
LIN {X 0,Y 424.349,Z 382.552,A -85,B 0,C 180,E1 -9635.703,E2 -9635.703} C_VEL
LIN {X 0,Y 424.555,Z 377.74,A -85,B 0,C 180,E1 -9637.61,E2 -9637.61} C_VEL
LIN {X 0,Y 424.982,Z 371.294,A -85,B 0,C 180,E1 -9639.519,E2 -9639.519} C_VEL
LIN {X 0,Y 425.478,Z 364.115,A -85,B 0,C 180,E1 -9641.191,E2 -9641.191} C_VEL
LIN {X 0,Y 426.193,Z 356.589,A -85,B 0,C 180,E1 -9642.621,E2 -9642.621} C_VEL
LIN {X 0,Y 426.715,Z 349.177,A -85,B 0,C 180,E1 -9643.816,E2 -9643.816} C_VEL
LIN {X 0,Y 427.691,Z 338.547,A -85,B 0,C 180,E1 -9645.243,E2 -9645.243} C_VEL
LIN {X 0,Y 428.554,Z 327.799,A -85,B 0,C 180,E1 -9646.433,E2 -9646.433} C_VEL
LIN {X 0,Y 429.528,Z 316.035,A -85,B 0,C 180,E1 -9647.497,E2 -9647.497} C_VEL
LIN {X 0,Y 430.358,Z 304.005,A -85,B 0,C 180,E1 -9648.379,E2 -9648.379} C_VEL
LIN {X 0,Y 431.069,Z 290.741,A -85,B 0,C 180,E1 -9649.147,E2 -9649.147} C_VEL
LIN {X 0,Y 431.19,Z 286.037,A -85,B 0,C 180,E1 -9649.373,E2 -9649.373} C_VEL
LIN {X 0,Y 428.107,Z 272.386,A -85,B 0,C 180,E1 -9650.07,E2 -9650.07} C_VEL
LIN {X 0,Y 424.523,Z 259.124,A -85,B 0,C 180,E1 -9650.629,E2 -9650.629} C_VEL
LIN {X 0,Y 424.632,Z 255.108,A -85,B 0,C 180,E1 -9653.405,E2 -9653.405} C_VEL
LIN {X 0,Y 424.765,Z 250.46,A -85,B 0,C 180,E1 -9656.688,E2 -9656.688} C_VEL
LIN {X 0,Y 424.946,Z 246.283,A -85,B 0,C 180,E1 -9659.746,E2 -9659.746} C_VEL
LIN {X 0,Y 425.147,Z 241.934,A -85,B 0,C 180,E1 -9663.06,E2 -9663.06} C_VEL
LIN {X 0,Y 425.34,Z 238.247,A -85,B 0,C 180,E1 -9665.939,E2 -9665.939} C_VEL
LIN {X 0,Y 425.349,Z 234.416,A -85,B 0,C 180,E1 -9669.052,E2 -9669.052} C_VEL
LIN {X 0,Y 425.244,Z 233.146,A -85,B 0,C 180,E1 -9670.132,E2 -9670.132} C_VEL
LIN {X 0,Y 425.26,Z 233.141,A -85,B 0,C 180,E1 -9673.351,E2 -9673.351} C_VEL
LIN {X 0,Y 425.261,Z 233.141,A -85,B 0,C 180,E1 -9676.044,E2 -9676.044} C_VEL
LIN {X 0,Y 425.257,Z 233.141,A -85,B 0,C 180,E1 -9679.484,E2 -9679.484} C_VEL
LIN {X 0,Y 425.279,Z 233.136,A -85,B 0,C 180,E1 -9682.489,E2 -9682.489} C_VEL
LIN {X 0,Y 425.308,Z 233.134,A -85,B 0,C 180,E1 -9685.817,E2 -9685.817} C_VEL
LIN {X 0,Y 425.293,Z 233.137,A -85,B 0,C 180,E1 -9689.239,E2 -9689.239} C_VEL
LIN {X 0,Y 425.351,Z 233.129,A -85,B 0,C 180,E1 -9692.442,E2 -9692.442} C_VEL
LIN {X 0,Y 425.351,Z 233.125,A -85,B 0,C 180,E1 -9695.602,E2 -9695.602} C_VEL
LIN {X 0,Y 425.296,Z 233.134,A -85,B 0,C 180,E1 -9698.682,E2 -9698.682} C_VEL
LIN {X 0,Y 425.332,Z 233.128,A -85,B 0,C 180,E1 -9701.703,E2 -9701.703} C_VEL
LIN {X 0,Y 425.35,Z 233.125,A -85,B 0,C 180,E1 -9704.671,E2 -9704.671} C_VEL
LIN {X 0,Y 425.415,Z 233.118,A -85,B 0,C 180,E1 -9707.598,E2 -9707.598} C_VEL
LIN {X 0,Y 425.411,Z 233.118,A -85,B 0,C 180,E1 -9711.449,E2 -9711.449} C_VEL
LIN {X 0,Y 425.55,Z 233.099,A -85,B 0,C 180,E1 -9714.313,E2 -9714.313} C_VEL
LIN {X 0,Y 425.574,Z 233.099,A -85,B 0,C 180,E1 -9718.107,E2 -9718.107} C_VEL
LIN {X 0,Y 425.533,Z 233.103,A -85,B 0,C 180,E1 -9720.946,E2 -9720.946} C_VEL
LIN {X 0,Y 425.548,Z 233.1,A -85,B 0,C 180,E1 -9722.84,E2 -9722.84} C_VEL
LIN {X 0,Y 425.535,Z 233.102,A -85,B 0,C 180,E1 -9725.687,E2 -9725.687} C_VEL
LIN {X 0,Y 425.409,Z 233.12,A -85,B 0,C 180,E1 -9728.551,E2 -9728.551} C_VEL
LIN {X 0,Y 425.415,Z 233.117,A -85,B 0,C 180,E1 -9732.402,E2 -9732.402} C_VEL
LIN {X 0,Y 425.39,Z 233.124,A -85,B 0,C 180,E1 -9736.312,E2 -9736.312} C_VEL
LIN {X 0,Y 425.331,Z 233.132,A -85,B 0,C 180,E1 -9739.635,E2 -9739.635} C_VEL
LIN {X 0,Y 425.29,Z 233.135,A -85,B 0,C 180,E1 -9742.339,E2 -9742.339} C_VEL
LIN {X 0,Y 425.321,Z 233.129,A -85,B 0,C 180,E1 -9744.657,E2 -9744.657} C_VEL
LIN {X 0,Y 425.254,Z 233.141,A -85,B 0,C 180,E1 -9747.564,E2 -9747.564} C_VEL
LIN {X 0,Y 425.292,Z 233.136,A -85,B 0,C 180,E1 -9750.761,E2 -9750.761} C_VEL
LIN {X 0,Y 425.313,Z 233.135,A -85,B 0,C 180,E1 -9754.288,E2 -9754.288} C_VEL
LIN {X 0,Y 425.28,Z 233.138,A -85,B 0,C 180,E1 -9757.694,E2 -9757.694} C_VEL
LIN {X 0,Y 425.282,Z 233.139,A -85,B 0,C 180,E1 -9760.52,E2 -9760.52} C_VEL
LIN {X 0,Y 425.259,Z 233.144,A -85,B 0,C 180,E1 -9763.351,E2 -9763.351} C_VEL
LIN {X 0,Y 425.315,Z 233.156,A -85,B 0,C 180,E1 -9766.47,E2 -9766.47} C_VEL
LIN {X 0,Y 425.955,Z 237.492,A -85,B 0,C 180,E1 -9769.374,E2 -9769.374} C_VEL
LIN {X 0,Y 426.236,Z 240.364,A -85,B 0,C 180,E1 -9771.203,E2 -9771.203} C_VEL
LIN {X 0,Y 426.07,Z 244.888,A -85,B 0,C 180,E1 -9773.925,E2 -9773.925} C_VEL
LIN {X 0,Y 425.729,Z 250.817,A -85,B 0,C 180,E1 -9777.343,E2 -9777.343} C_VEL
LIN {X 0,Y 425.439,Z 256.128,A -85,B 0,C 180,E1 -9780.292,E2 -9780.292} C_VEL
LIN {X 0,Y 425.19,Z 261.483,A -85,B 0,C 180,E1 -9783.198,E2 -9783.198} C_VEL
LIN {X 0,Y 424.823,Z 267.885,A -85,B 0,C 180,E1 -9786.606,E2 -9786.606} C_VEL
LIN {X 0,Y 424.601,Z 273.286,A -85,B 0,C 180,E1 -9789.424,E2 -9789.424} C_VEL
LIN {X 0,Y 428.145,Z 288.543,A -85,B 0,C 180,E1 -9790.007,E2 -9790.007} C_VEL
LIN {X 0,Y 430.549,Z 301.827,A -85,B 0,C 180,E1 -9790.66,E2 -9790.66} C_VEL
LIN {X 0,Y 430.884,Z 305.397,A -85,B 0,C 180,E1 -9790.847,E2 -9790.847} C_VEL
LIN {X 0,Y 430.09,Z 318.505,A -85,B 0,C 180,E1 -9791.585,E2 -9791.585} C_VEL
LIN {X 0,Y 429.129,Z 331.053,A -85,B 0,C 180,E1 -9792.486,E2 -9792.486} C_VEL
LIN {X 0,Y 428.207,Z 342.962,A -85,B 0,C 180,E1 -9793.553,E2 -9793.553} C_VEL
LIN {X 0,Y 427.293,Z 353.841,A -85,B 0,C 180,E1 -9794.742,E2 -9794.742} C_VEL
LIN {X 0,Y 426.419,Z 364.594,A -85,B 0,C 180,E1 -9796.173,E2 -9796.173} C_VEL
LIN {X 0,Y 425.728,Z 373.474,A -85,B 0,C 180,E1 -9797.607,E2 -9797.607} C_VEL
LIN {X 0,Y 425.065,Z 381.985,A -85,B 0,C 180,E1 -9799.28,E2 -9799.28} C_VEL
LIN {X 0,Y 424.607,Z 388.845,A -85,B 0,C 180,E1 -9800.953,E2 -9800.953} C_VEL
LIN {X 0,Y 424.348,Z 393.574,A -85,B 0,C 180,E1 -9802.386,E2 -9802.386} C_VEL
LIN {X 0,Y 424.247,Z 397.126,A -85,B 0,C 180,E1 -9803.694,E2 -9803.694} C_VEL
LIN {X 0,Y 424.171,Z 400.358,A -85,B 0,C 180,E1 -9805.248,E2 -9805.248} C_VEL
LIN {X 0,Y 424.082,Z 403.06,A -85,B 0,C 180,E1 -9807.15,E2 -9807.15} C_VEL
LIN {X 0,Y 424.066,Z 404.399,A -85,B 0,C 180,E1 -9809.05,E2 -9809.05} C_VEL
LIN {X 0,Y 424.066,Z 404.398,A -85,B 0,C 180,E1 -9810.95,E2 -9810.95} C_VEL
LIN {X 0,Y 424.082,Z 403.059,A -85,B 0,C 180,E1 -9812.85,E2 -9812.85} C_VEL
LIN {X 0,Y 424.171,Z 400.356,A -85,B 0,C 180,E1 -9814.752,E2 -9814.752} C_VEL
LIN {X 0,Y 424.297,Z 396.212,A -85,B 0,C 180,E1 -9816.658,E2 -9816.658} C_VEL
LIN {X 0,Y 424.516,Z 390.504,A -85,B 0,C 180,E1 -9818.569,E2 -9818.569} C_VEL
LIN {X 0,Y 424.909,Z 384.071,A -85,B 0,C 180,E1 -9820.242,E2 -9820.242} C_VEL
LIN {X 0,Y 425.554,Z 376.082,A -85,B 0,C 180,E1 -9821.914,E2 -9821.914} C_VEL
LIN {X 0,Y 426.166,Z 367.725,A -85,B 0,C 180,E1 -9823.349,E2 -9823.349} C_VEL
LIN {X 0,Y 426.973,Z 357.665,A -85,B 0,C 180,E1 -9824.781,E2 -9824.781} C_VEL
LIN {X 0,Y 427.891,Z 346.446,A -85,B 0,C 180,E1 -9826.091,E2 -9826.091} C_VEL
LIN {X 0,Y 428.812,Z 335.287,A -85,B 0,C 180,E1 -9827.158,E2 -9827.158} C_VEL
LIN {X 0,Y 429.768,Z 323.136,A -85,B 0,C 180,E1 -9828.102,E2 -9828.102} C_VEL
LIN {X 0,Y 430.572,Z 309.994,A -85,B 0,C 180,E1 -9828.911,E2 -9828.911} C_VEL
LIN {X 0,Y 430.804,Z 302.967,A -85,B 0,C 180,E1 -9829.269,E2 -9829.269} C_VEL
LIN {X 0,Y 428.115,Z 288.521,A -85,B 0,C 180,E1 -9829.989,E2 -9829.989} C_VEL
LIN {X 0,Y 424.982,Z 275.295,A -85,B 0,C 180,E1 -9830.505,E2 -9830.505} C_VEL
LIN {X 0,Y 424.602,Z 273.241,A -85,B 0,C 180,E1 -9830.593,E2 -9830.593} C_VEL
LIN {X 0,Y 424.82,Z 267.865,A -85,B 0,C 180,E1 -9833.393,E2 -9833.393} C_VEL
LIN {X 0,Y 425.194,Z 261.466,A -85,B 0,C 180,E1 -9836.803,E2 -9836.803} C_VEL
LIN {X 0,Y 425.431,Z 256.112,A -85,B 0,C 180,E1 -9839.709,E2 -9839.709} C_VEL
LIN {X 0,Y 425.732,Z 250.167,A -85,B 0,C 180,E1 -9843.009,E2 -9843.009} C_VEL
LIN {X 0,Y 426.073,Z 244.852,A -85,B 0,C 180,E1 -9846.075,E2 -9846.075} C_VEL
LIN {X 0,Y 426.236,Z 240.341,A -85,B 0,C 180,E1 -9848.797,E2 -9848.797} C_VEL
LIN {X 0,Y 425.804,Z 236.422,A -85,B 0,C 180,E1 -9851.316,E2 -9851.316} C_VEL
LIN {X 0,Y 425.29,Z 233.138,A -85,B 0,C 180,E1 -9853.616,E2 -9853.616} C_VEL
LIN {X 0,Y 425.258,Z 233.141,A -85,B 0,C 180,E1 -9856.649,E2 -9856.649} C_VEL
LIN {X 0,Y 425.287,Z 233.136,A -85,B 0,C 180,E1 -9859.873,E2 -9859.873} C_VEL
LIN {X 0,Y 425.277,Z 233.14,A -85,B 0,C 180,E1 -9862.489,E2 -9862.489} C_VEL
LIN {X 0,Y 425.308,Z 233.136,A -85,B 0,C 180,E1 -9865.817,E2 -9865.817} C_VEL
LIN {X 0,Y 425.291,Z 233.137,A -85,B 0,C 180,E1 -9869.239,E2 -9869.239} C_VEL
LIN {X 0,Y 425.27,Z 233.14,A -85,B 0,C 180,E1 -9872.437,E2 -9872.437} C_VEL
LIN {X 0,Y 425.347,Z 233.13,A -85,B 0,C 180,E1 -9875.602,E2 -9875.602} C_VEL
LIN {X 0,Y 425.294,Z 233.136,A -85,B 0,C 180,E1 -9878.682,E2 -9878.682} C_VEL
LIN {X 0,Y 425.321,Z 233.13,A -85,B 0,C 180,E1 -9881.702,E2 -9881.702} C_VEL
LIN {X 0,Y 425.35,Z 233.125,A -85,B 0,C 180,E1 -9884.671,E2 -9884.671} C_VEL
LIN {X 0,Y 425.414,Z 233.118,A -85,B 0,C 180,E1 -9887.598,E2 -9887.598} C_VEL
LIN {X 0,Y 425.408,Z 233.119,A -85,B 0,C 180,E1 -9891.449,E2 -9891.449} C_VEL
LIN {X 0,Y 425.533,Z 233.102,A -85,B 0,C 180,E1 -9894.313,E2 -9894.313} C_VEL
LIN {X 0,Y 425.575,Z 233.099,A -85,B 0,C 180,E1 -9898.107,E2 -9898.107} C_VEL
LIN {X 0,Y 425.697,Z 233.086,A -85,B 0,C 180,E1 -9900,E2 -9900} C_VEL
LIN {X 0,Y 425.537,Z 233.103,A -85,B 0,C 180,E1 -9902.84,E2 -9902.84} C_VEL
LIN {X 0,Y 425.525,Z 233.106,A -85,B 0,C 180,E1 -9906.639,E2 -9906.639} C_VEL
LIN {X 0,Y 425.402,Z 233.121,A -85,B 0,C 180,E1 -9909.509,E2 -9909.509} C_VEL
LIN {X 0,Y 425.395,Z 233.124,A -85,B 0,C 180,E1 -9912.904,E2 -9912.904} C_VEL
LIN {X 0,Y 425.364,Z 233.125,A -85,B 0,C 180,E1 -9916.605,E2 -9916.605} C_VEL
LIN {X 0,Y 425.331,Z 233.13,A -85,B 0,C 180,E1 -9919.636,E2 -9919.636} C_VEL
LIN {X 0,Y 425.289,Z 233.134,A -85,B 0,C 180,E1 -9922.339,E2 -9922.339} C_VEL
LIN {X 0,Y 425.293,Z 233.133,A -85,B 0,C 180,E1 -9925.446,E2 -9925.446} C_VEL
LIN {X 0,Y 425.35,Z 233.129,A -85,B 0,C 180,E1 -9927.558,E2 -9927.558} C_VEL
LIN {X 0,Y 425.289,Z 233.136,A -85,B 0,C 180,E1 -9930.816,E2 -9930.816} C_VEL
LIN {X 0,Y 425.311,Z 233.133,A -85,B 0,C 180,E1 -9934.288,E2 -9934.288} C_VEL
LIN {X 0,Y 425.278,Z 233.136,A -85,B 0,C 180,E1 -9937.695,E2 -9937.695} C_VEL
LIN {X 0,Y 425.256,Z 233.141,A -85,B 0,C 180,E1 -9940.516,E2 -9940.516} C_VEL
LIN {X 0,Y 425.26,Z 233.141,A -85,B 0,C 180,E1 -9943.956,E2 -9943.956} C_VEL
LIN {X 0,Y 425.275,Z 233.139,A -85,B 0,C 180,E1 -9947.347,E2 -9947.347} C_VEL
LIN {X 0,Y 425.263,Z 233.14,A -85,B 0,C 180,E1 -9949.87,E2 -9949.87} C_VEL
LIN {X 0,Y 425.381,Z 236.134,A -85,B 0,C 180,E1 -9952.471,E2 -9952.471} C_VEL
LIN {X 0,Y 425.261,Z 240.216,A -85,B 0,C 180,E1 -9955.722,E2 -9955.722} C_VEL
LIN {X 0,Y 425.004,Z 244.882,A -85,B 0,C 180,E1 -9959.304,E2 -9959.304} C_VEL
LIN {X 0,Y 424.793,Z 249.057,A -85,B 0,C 180,E1 -9962.403,E2 -9962.403} C_VEL
LIN {X 0,Y 424.717,Z 253.494,A -85,B 0,C 180,E1 -9965.563,E2 -9965.563} C_VEL
LIN {X 0,Y 424.529,Z 258.662,A -85,B 0,C 180,E1 -9969.15,E2 -9969.15} C_VEL
LIN {X 0,Y 424.54,Z 259.155,A -85,B 0,C 180,E1 -9969.491,E2 -9969.491} C_VEL
LIN {X 0,Y 428.654,Z 274.653,A -85,B 0,C 180,E1 -9970.13,E2 -9970.13} C_VEL
LIN {X 0,Y 431.161,Z 286.137,A -85,B 0,C 180,E1 -9970.727,E2 -9970.727} C_VEL
LIN {X 0,Y 430.646,Z 298.55,A -85,B 0,C 180,E1 -9971.376,E2 -9971.376} C_VEL
LIN {X 0,Y 429.831,Z 311.856,A -85,B 0,C 180,E1 -9972.27,E2 -9972.27} C_VEL
LIN {X 0,Y 428.82,Z 324.44,A -85,B 0,C 180,E1 -9973.333,E2 -9973.333} C_VEL
LIN {X 0,Y 427.92,Z 335.797,A -85,B 0,C 180,E1 -9974.521,E2 -9974.521} C_VEL
LIN {X 0,Y 427.072,Z 345.211,A -85,B 0,C 180,E1 -9975.709,E2 -9975.709} C_VEL
LIN {X 0,Y 426.306,Z 354.664,A -85,B 0,C 180,E1 -9977.141,E2 -9977.141} C_VEL
LIN {X 0,Y 425.604,Z 362.498,A -85,B 0,C 180,E1 -9978.571,E2 -9978.571} C_VEL
LIN {X 0,Y 425.141,Z 369.01,A -85,B 0,C 180,E1 -9980.004,E2 -9980.004} C_VEL
LIN {X 0,Y 424.76,Z 374.416,A -85,B 0,C 180,E1 -9981.436,E2 -9981.436} C_VEL
LIN {X 0,Y 424.456,Z 380.098,A -85,B 0,C 180,E1 -9983.344,E2 -9983.344} C_VEL
LIN {X 0,Y 424.227,Z 384.228,A -85,B 0,C 180,E1 -9985.249,E2 -9985.249} C_VEL
LIN {X 0,Y 424.174,Z 386.929,A -85,B 0,C 180,E1 -9987.151,E2 -9987.151} C_VEL
LIN {X 0,Y 424.068,Z 388.286,A -85,B 0,C 180,E1 -9989.05,E2 -9989.05} C_VEL
LIN {X 0,Y 424.05,Z 388.422,A -85,B 0,C 180,E1 -9990.301,E2 -9990.301} C_VEL
LIN {X 0,Y 423.374,Z 388.273,A -85,B 0,C 180,E1 -9991.095,E2 -9991.095} C_VEL
LIN {X 0,Y 420.506,Z 387.531,A -85,B 0,C 180,E1 -9992.381,E2 -9992.381} C_VEL
LIN {X 0,Y 418.123,Z 386.545,A -85,B 0,C 180,E1 -9993.414,E2 -9993.414} C_VEL
LIN {X 0,Y 417.153,Z 385.512,A -85,B 0,C 180,E1 -9994.206,E2 -9994.206} C_VEL
LIN {X 0,Y 417.104,Z 385.086,A -85,B 0,C 180,E1 -9994.473,E2 -9994.473} C_VEL
LIN {X 0,Y 417.352,Z 381.107,A -85,B 0,C 180,E1 -9996.519,E2 -9996.519} C_VEL
LIN {X 0,Y 417.592,Z 376.456,A -85,B 0,C 180,E1 -9998.225,E2 -9998.225} C_VEL
LIN {X 0,Y 417.955,Z 371.427,A -85,B 0,C 180,E1 -9999.681,E2 -9999.681} C_VEL
LIN {X 0,Y 418.475,Z 364.249,A -85,B 0,C 180,E1 -10001.381,E2 -10001.381} C_VEL
LIN {X 0,Y 419.236,Z 356.77,A -85,B 0,C 180,E1 -10002.825,E2 -10002.825} C_VEL
LIN {X 0,Y 419.954,Z 347.846,A -85,B 0,C 180,E1 -10004.266,E2 -10004.266} C_VEL
LIN {X 0,Y 421.007,Z 336.732,A -85,B 0,C 180,E1 -10005.74,E2 -10005.74} C_VEL
LIN {X 0,Y 421.982,Z 325.562,A -85,B 0,C 180,E1 -10006.945,E2 -10006.945} C_VEL
LIN {X 0,Y 422.966,Z 313.199,A -85,B 0,C 180,E1 -10008.028,E2 -10008.028} C_VEL
LIN {X 0,Y 423.784,Z 301.085,A -85,B 0,C 180,E1 -10008.881,E2 -10008.881} C_VEL
LIN {X 0,Y 424.52,Z 288.095,A -85,B 0,C 180,E1 -10009.596,E2 -10009.596} C_VEL
LIN {X 0,Y 421.962,Z 276.001,A -85,B 0,C 180,E1 -10010.253,E2 -10010.253} C_VEL
LIN {X 0,Y 418.164,Z 261.961,A -85,B 0,C 180,E1 -10010.872,E2 -10010.872} C_VEL
LIN {X 0,Y 417.467,Z 259.255,A -85,B 0,C 180,E1 -10010.994,E2 -10010.994} C_VEL
LIN {X 0,Y 417.647,Z 254.038,A -85,B 0,C 180,E1 -10014.674,E2 -10014.674} C_VEL
LIN {X 0,Y 417.772,Z 249.305,A -85,B 0,C 180,E1 -10018.102,E2 -10018.102} C_VEL
LIN {X 0,Y 417.992,Z 244.942,A -85,B 0,C 180,E1 -10021.415,E2 -10021.415} C_VEL
LIN {X 0,Y 418.252,Z 240.561,A -85,B 0,C 180,E1 -10024.842,E2 -10024.842} C_VEL
LIN {X 0,Y 418.329,Z 236.869,A -85,B 0,C 180,E1 -10027.851,E2 -10027.851} C_VEL
LIN {X 0,Y 418.245,Z 234.688,A -85,B 0,C 180,E1 -10029.683,E2 -10029.683} C_VEL
LIN {X 0,Y 418.214,Z 234.021,A -85,B 0,C 180,E1 -10030.949,E2 -10030.949} C_VEL
LIN {X 0,Y 418.212,Z 234.017,A -85,B 0,C 180,E1 -10033.729,E2 -10033.729} C_VEL
LIN {X 0,Y 418.205,Z 234.021,A -85,B 0,C 180,E1 -10036.448,E2 -10036.448} C_VEL
LIN {X 0,Y 418.213,Z 234.017,A -85,B 0,C 180,E1 -10039.132,E2 -10039.132} C_VEL
LIN {X 0,Y 418.241,Z 234.015,A -85,B 0,C 180,E1 -10042.776,E2 -10042.776} C_VEL
LIN {X 0,Y 418.25,Z 234.012,A -85,B 0,C 180,E1 -10046.323,E2 -10046.323} C_VEL
LIN {X 0,Y 418.247,Z 234.012,A -85,B 0,C 180,E1 -10049.728,E2 -10049.728} C_VEL
LIN {X 0,Y 418.307,Z 234.004,A -85,B 0,C 180,E1 -10053.023,E2 -10053.023} C_VEL
LIN {X 0,Y 418.278,Z 234.007,A -85,B 0,C 180,E1 -10056.218,E2 -10056.218} C_VEL
LIN {X 0,Y 418.253,Z 234.01,A -85,B 0,C 180,E1 -10059.337,E2 -10059.337} C_VEL
LIN {X 0,Y 418.288,Z 234.008,A -85,B 0,C 180,E1 -10062.396,E2 -10062.396} C_VEL
LIN {X 0,Y 418.305,Z 234.007,A -85,B 0,C 180,E1 -10065.403,E2 -10065.403} C_VEL
LIN {X 0,Y 418.318,Z 234.003,A -85,B 0,C 180,E1 -10068.369,E2 -10068.369} C_VEL
LIN {X 0,Y 418.468,Z 233.984,A -85,B 0,C 180,E1 -10072.278,E2 -10072.278} C_VEL
LIN {X 0,Y 418.508,Z 233.977,A -85,B 0,C 180,E1 -10074.217,E2 -10074.217} C_VEL
LIN {X 0,Y 418.543,Z 233.974,A -85,B 0,C 180,E1 -10078.075,E2 -10078.075} C_VEL
LIN {X 0,Y 418.494,Z 233.979,A -85,B 0,C 180,E1 -10080.962,E2 -10080.962} C_VEL
LIN {X 0,Y 418.503,Z 233.978,A -85,B 0,C 180,E1 -10082.888,E2 -10082.888} C_VEL
LIN {X 0,Y 418.492,Z 233.98,A -85,B 0,C 180,E1 -10085.783,E2 -10085.783} C_VEL
LIN {X 0,Y 418.379,Z 233.995,A -85,B 0,C 180,E1 -10088.695,E2 -10088.695} C_VEL
LIN {X 0,Y 418.318,Z 234.003,A -85,B 0,C 180,E1 -10091.631,E2 -10091.631} C_VEL
LIN {X 0,Y 418.307,Z 234.006,A -85,B 0,C 180,E1 -10094.597,E2 -10094.597} C_VEL
LIN {X 0,Y 418.281,Z 234.008,A -85,B 0,C 180,E1 -10097.604,E2 -10097.604} C_VEL
LIN {X 0,Y 418.252,Z 234.011,A -85,B 0,C 180,E1 -10100.663,E2 -10100.663} C_VEL
LIN {X 0,Y 418.276,Z 234.007,A -85,B 0,C 180,E1 -10103.782,E2 -10103.782} C_VEL
LIN {X 0,Y 418.211,Z 234.015,A -85,B 0,C 180,E1 -10107.043,E2 -10107.043} C_VEL
LIN {X 0,Y 418.243,Z 234.012,A -85,B 0,C 180,E1 -10110.272,E2 -10110.272} C_VEL
LIN {X 0,Y 418.251,Z 234.011,A -85,B 0,C 180,E1 -10113.677,E2 -10113.677} C_VEL
LIN {X 0,Y 418.241,Z 234.017,A -85,B 0,C 180,E1 -10117.224,E2 -10117.224} C_VEL
LIN {X 0,Y 418.248,Z 234.012,A -85,B 0,C 180,E1 -10119.682,E2 -10119.682} C_VEL
LIN {X 0,Y 418.232,Z 234.019,A -85,B 0,C 180,E1 -10122.321,E2 -10122.321} C_VEL
LIN {X 0,Y 418.257,Z 234.013,A -85,B 0,C 180,E1 -10126.155,E2 -10126.155} C_VEL
LIN {X 0,Y 418.898,Z 238.322,A -85,B 0,C 180,E1 -10129.132,E2 -10129.132} C_VEL
LIN {X 0,Y 419.209,Z 242.243,A -85,B 0,C 180,E1 -10131.662,E2 -10131.662} C_VEL
LIN {X 0,Y 419.02,Z 246.167,A -85,B 0,C 180,E1 -10134.053,E2 -10134.053} C_VEL
LIN {X 0,Y 418.668,Z 252.076,A -85,B 0,C 180,E1 -10137.509,E2 -10137.509} C_VEL
LIN {X 0,Y 418.354,Z 258.057,A -85,B 0,C 180,E1 -10140.875,E2 -10140.875} C_VEL
LIN {X 0,Y 418.011,Z 263.858,A -85,B 0,C 180,E1 -10144.078,E2 -10144.078} C_VEL
LIN {X 0,Y 417.67,Z 270.652,A -85,B 0,C 180,E1 -10147.739,E2 -10147.739} C_VEL
LIN {X 0,Y 417.567,Z 273.121,A -85,B 0,C 180,E1 -10149.043,E2 -10149.043} C_VEL
LIN {X 0,Y 421.569,Z 290.338,A -85,B 0,C 180,E1 -10149.748,E2 -10149.748} C_VEL
LIN {X 0,Y 423.873,Z 303.529,A -85,B 0,C 180,E1 -10150.431,E2 -10150.431} C_VEL
LIN {X 0,Y 424.048,Z 307.36,A -85,B 0,C 180,E1 -10150.642,E2 -10150.642} C_VEL
LIN {X 0,Y 423.223,Z 320.11,A -85,B 0,C 180,E1 -10151.398,E2 -10151.398} C_VEL
LIN {X 0,Y 422.226,Z 332.35,A -85,B 0,C 180,E1 -10152.315,E2 -10152.315} C_VEL
LIN {X 0,Y 421.268,Z 344.006,A -85,B 0,C 180,E1 -10153.399,E2 -10153.399} C_VEL
LIN {X 0,Y 420.388,Z 353.708,A -85,B 0,C 180,E1 -10154.485,E2 -10154.485} C_VEL
LIN {X 0,Y 419.485,Z 364.46,A -85,B 0,C 180,E1 -10155.94,E2 -10155.94} C_VEL
LIN {X 0,Y 418.728,Z 373.34,A -85,B 0,C 180,E1 -10157.397,E2 -10157.397} C_VEL
LIN {X 0,Y 418.029,Z 381.85,A -85,B 0,C 180,E1 -10159.097,E2 -10159.097} C_VEL
LIN {X 0,Y 417.559,Z 388.711,A -85,B 0,C 180,E1 -10160.799,E2 -10160.799} C_VEL
LIN {X 0,Y 417.295,Z 393.439,A -85,B 0,C 180,E1 -10162.257,E2 -10162.257} C_VEL
LIN {X 0,Y 417.168,Z 397.251,A -85,B 0,C 180,E1 -10163.704,E2 -10163.704} C_VEL
LIN {X 0,Y 417.078,Z 400.224,A -85,B 0,C 180,E1 -10165.167,E2 -10165.167} C_VEL
LIN {X 0,Y 416.979,Z 402.926,A -85,B 0,C 180,E1 -10167.102,E2 -10167.102} C_VEL
LIN {X 0,Y 416.99,Z 404.265,A -85,B 0,C 180,E1 -10169.034,E2 -10169.034} C_VEL
LIN {X 0,Y 416.99,Z 404.264,A -85,B 0,C 180,E1 -10170.966,E2 -10170.966} C_VEL
LIN {X 0,Y 416.979,Z 402.924,A -85,B 0,C 180,E1 -10172.898,E2 -10172.898} C_VEL
LIN {X 0,Y 417.077,Z 400.221,A -85,B 0,C 180,E1 -10174.833,E2 -10174.833} C_VEL
LIN {X 0,Y 417.228,Z 396.076,A -85,B 0,C 180,E1 -10176.772,E2 -10176.772} C_VEL
LIN {X 0,Y 417.458,Z 390.367,A -85,B 0,C 180,E1 -10178.715,E2 -10178.715} C_VEL
LIN {X 0,Y 417.858,Z 383.934,A -85,B 0,C 180,E1 -10180.417,E2 -10180.417} C_VEL
LIN {X 0,Y 418.567,Z 375.945,A -85,B 0,C 180,E1 -10182.115,E2 -10182.115} C_VEL
LIN {X 0,Y 419.209,Z 367.587,A -85,B 0,C 180,E1 -10183.574,E2 -10183.574} C_VEL
LIN {X 0,Y 420.058,Z 357.527,A -85,B 0,C 180,E1 -10185.03,E2 -10185.03} C_VEL
LIN {X 0,Y 421.044,Z 346.308,A -85,B 0,C 180,E1 -10186.36,E2 -10186.36} C_VEL
LIN {X 0,Y 422.006,Z 335.148,A -85,B 0,C 180,E1 -10187.444,E2 -10187.444} C_VEL
LIN {X 0,Y 423.016,Z 322.997,A -85,B 0,C 180,E1 -10188.401,E2 -10188.401} C_VEL
LIN {X 0,Y 423.83,Z 310.166,A -85,B 0,C 180,E1 -10189.206,E2 -10189.206} C_VEL
LIN {X 0,Y 423.957,Z 303.46,A -85,B 0,C 180,E1 -10189.562,E2 -10189.562} C_VEL
LIN {X 0,Y 421.303,Z 289.13,A -85,B 0,C 180,E1 -10190.3,E2 -10190.3} C_VEL
LIN {X 0,Y 417.772,Z 274.531,A -85,B 0,C 180,E1 -10190.889,E2 -10190.889} C_VEL
LIN {X 0,Y 417.566,Z 273.104,A -85,B 0,C 180,E1 -10190.957,E2 -10190.957} C_VEL
LIN {X 0,Y 417.767,Z 267.742,A -85,B 0,C 180,E1 -10193.813,E2 -10193.813} C_VEL
LIN {X 0,Y 418.15,Z 261.827,A -85,B 0,C 180,E1 -10197.027,E2 -10197.027} C_VEL
LIN {X 0,Y 418.42,Z 256,A -85,B 0,C 180,E1 -10200.258,E2 -10200.258} C_VEL
LIN {X 0,Y 418.751,Z 250.074,A -85,B 0,C 180,E1 -10203.631,E2 -10203.631} C_VEL
LIN {X 0,Y 419.098,Z 245.377,A -85,B 0,C 180,E1 -10206.397,E2 -10206.397} C_VEL
LIN {X 0,Y 419.217,Z 242.213,A -85,B 0,C 180,E1 -10208.337,E2 -10208.337} C_VEL
LIN {X 0,Y 418.896,Z 238.135,A -85,B 0,C 180,E1 -10210.976,E2 -10210.976} C_VEL
LIN {X 0,Y 418.257,Z 234.012,A -85,B 0,C 180,E1 -10213.845,E2 -10213.845} C_VEL
LIN {X 0,Y 418.241,Z 234.015,A -85,B 0,C 180,E1 -10217.767,E2 -10217.767} C_VEL
LIN {X 0,Y 418.25,Z 234.013,A -85,B 0,C 180,E1 -10220.62,E2 -10220.62} C_VEL
LIN {X 0,Y 418.243,Z 234.015,A -85,B 0,C 180,E1 -10223.976,E2 -10223.976} C_VEL
LIN {X 0,Y 418.259,Z 234.012,A -85,B 0,C 180,E1 -10227.156,E2 -10227.156} C_VEL
LIN {X 0,Y 418.26,Z 234.013,A -85,B 0,C 180,E1 -10230.838,E2 -10230.838} C_VEL
LIN {X 0,Y 418.236,Z 234.016,A -85,B 0,C 180,E1 -10234.094,E2 -10234.094} C_VEL
LIN {X 0,Y 418.233,Z 234.016,A -85,B 0,C 180,E1 -10237.264,E2 -10237.264} C_VEL
LIN {X 0,Y 418.284,Z 234.009,A -85,B 0,C 180,E1 -10240.364,E2 -10240.364} C_VEL
LIN {X 0,Y 418.317,Z 234.002,A -85,B 0,C 180,E1 -10243.405,E2 -10243.405} C_VEL
LIN {X 0,Y 418.348,Z 234.001,A -85,B 0,C 180,E1 -10246.999,E2 -10246.999} C_VEL
LIN {X 0,Y 418.337,Z 234.001,A -85,B 0,C 180,E1 -10250.329,E2 -10250.329} C_VEL
LIN {X 0,Y 418.445,Z 233.987,A -85,B 0,C 180,E1 -10253.248,E2 -10253.248} C_VEL
LIN {X 0,Y 418.333,Z 234.003,A -85,B 0,C 180,E1 -10255.182,E2 -10255.182} C_VEL
LIN {X 0,Y 418.544,Z 233.975,A -85,B 0,C 180,E1 -10258.076,E2 -10258.076} C_VEL
LIN {X 0,Y 418.666,Z 233.962,A -85,B 0,C 180,E1 -10260,E2 -10260} C_VEL
LIN {X 0,Y 418.492,Z 233.981,A -85,B 0,C 180,E1 -10262.888,E2 -10262.888} C_VEL
LIN {X 0,Y 418.489,Z 233.982,A -85,B 0,C 180,E1 -10266.751,E2 -10266.751} C_VEL
LIN {X 0,Y 418.342,Z 234.001,A -85,B 0,C 180,E1 -10269.671,E2 -10269.671} C_VEL
LIN {X 0,Y 418.348,Z 234.001,A -85,B 0,C 180,E1 -10273.001,E2 -10273.001} C_VEL
LIN {X 0,Y 418.315,Z 234.002,A -85,B 0,C 180,E1 -10276.736,E2 -10276.736} C_VEL
LIN {X 0,Y 418.273,Z 234.008,A -85,B 0,C 180,E1 -10279.79,E2 -10279.79} C_VEL
LIN {X 0,Y 418.233,Z 234.016,A -85,B 0,C 180,E1 -10282.737,E2 -10282.737} C_VEL
LIN {X 0,Y 418.27,Z 234.01,A -85,B 0,C 180,E1 -10285.904,E2 -10285.904} C_VEL
LIN {X 0,Y 418.266,Z 234.011,A -85,B 0,C 180,E1 -10289.162,E2 -10289.162} C_VEL
LIN {X 0,Y 418.258,Z 234.01,A -85,B 0,C 180,E1 -10292.844,E2 -10292.844} C_VEL
LIN {X 0,Y 418.246,Z 234.011,A -85,B 0,C 180,E1 -10296.238,E2 -10296.238} C_VEL
LIN {X 0,Y 418.211,Z 234.014,A -85,B 0,C 180,E1 -10299.687,E2 -10299.687} C_VEL
LIN {X 0,Y 418.214,Z 234.02,A -85,B 0,C 180,E1 -10302.319,E2 -10302.319} C_VEL
LIN {X 0,Y 418.237,Z 234.014,A -85,B 0,C 180,E1 -10305.109,E2 -10305.109} C_VEL
LIN {X 0,Y 418.239,Z 234.015,A -85,B 0,C 180,E1 -10307.767,E2 -10307.767} C_VEL
LIN {X 0,Y 418.216,Z 234.018,A -85,B 0,C 180,E1 -10309.132,E2 -10309.132} C_VEL
LIN {X 0,Y 418.287,Z 234.904,A -85,B 0,C 180,E1 -10310.614,E2 -10310.614} C_VEL
LIN {X 0,Y 418.315,Z 238.671,A -85,B 0,C 180,E1 -10313.749,E2 -10313.749} C_VEL
LIN {X 0,Y 418.149,Z 241.877,A -85,B 0,C 180,E1 -10316.314,E2 -10316.314} C_VEL
LIN {X 0,Y 417.909,Z 246.249,A -85,B 0,C 180,E1 -10319.701,E2 -10319.701} C_VEL
LIN {X 0,Y 417.702,Z 250.806,A -85,B 0,C 180,E1 -10323.094,E2 -10323.094} C_VEL
LIN {X 0,Y 417.584,Z 255.093,A -85,B 0,C 180,E1 -10326.176,E2 -10326.176} C_VEL
LIN {X 0,Y 417.46,Z 259.289,A -85,B 0,C 180,E1 -10329.127,E2 -10329.127} C_VEL
LIN {X 0,Y 421.704,Z 274.821,A -85,B 0,C 180,E1 -10329.789,E2 -10329.789} C_VEL
LIN {X 0,Y 424.5,Z 287.906,A -85,B 0,C 180,E1 -10330.491,E2 -10330.491} C_VEL
LIN {X 0,Y 423.754,Z 301.542,A -85,B 0,C 180,E1 -10331.242,E2 -10331.242} C_VEL
LIN {X 0,Y 422.955,Z 313.575,A -85,B 0,C 180,E1 -10332.097,E2 -10332.097} C_VEL
LIN {X 0,Y 421.9,Z 325.854,A -85,B 0,C 180,E1 -10333.176,E2 -10333.176} C_VEL
LIN {X 0,Y 421.062,Z 335.936,A -85,B 0,C 180,E1 -10334.263,E2 -10334.263} C_VEL
LIN {X 0,Y 420.162,Z 345.35,A -85,B 0,C 180,E1 -10335.469,E2 -10335.469} C_VEL
LIN {X 0,Y 419.343,Z 354.803,A -85,B 0,C 180,E1 -10336.923,E2 -10336.923} C_VEL
LIN {X 0,Y 418.638,Z 362.635,A -85,B 0,C 180,E1 -10338.378,E2 -10338.378} C_VEL
LIN {X 0,Y 418.121,Z 369.147,A -85,B 0,C 180,E1 -10339.835,E2 -10339.835} C_VEL
LIN {X 0,Y 417.71,Z 374.553,A -85,B 0,C 180,E1 -10341.291,E2 -10341.291} C_VEL
LIN {X 0,Y 417.372,Z 380.234,A -85,B 0,C 180,E1 -10343.231,E2 -10343.231} C_VEL
LIN {X 0,Y 417.163,Z 384.363,A -85,B 0,C 180,E1 -10345.168,E2 -10345.168} C_VEL
LIN {X 0,Y 417.073,Z 387.065,A -85,B 0,C 180,E1 -10347.102,E2 -10347.102} C_VEL
LIN {X 0,Y 416.991,Z 388.42,A -85,B 0,C 180,E1 -10349.034,E2 -10349.034} C_VEL
LIN {X 0,Y 416.992,Z 388.456,A -85,B 0,C 180,E1 -10350.966,E2 -10350.966} C_VEL
LIN {X 0,Y 417.072,Z 387.17,A -85,B 0,C 180,E1 -10352.898,E2 -10352.898} C_VEL
LIN {X 0,Y 417.104,Z 385.086,A -85,B 0,C 180,E1 -10354.473,E2 -10354.473} C_VEL
LIN {X 0,Y 416.532,Z 383.794,A -85,B 0,C 180,E1 -10355.262,E2 -10355.262} C_VEL
LIN {X 0,Y 413.804,Z 381.33,A -85,B 0,C 180,E1 -10356.534,E2 -10356.534} C_VEL
LIN {X 0,Y 411.518,Z 378.924,A -85,B 0,C 180,E1 -10357.543,E2 -10357.543} C_VEL
LIN {X 0,Y 410.619,Z 376.769,A -85,B 0,C 180,E1 -10358.304,E2 -10358.304} C_VEL
LIN {X 0,Y 410.591,Z 375.976,A -85,B 0,C 180,E1 -10358.557,E2 -10358.557} C_VEL
LIN {X 0,Y 411.092,Z 369.668,A -85,B 0,C 180,E1 -10360.341,E2 -10360.341} C_VEL
LIN {X 0,Y 411.809,Z 362.013,A -85,B 0,C 180,E1 -10362.067,E2 -10362.067} C_VEL
LIN {X 0,Y 412.445,Z 353.753,A -85,B 0,C 180,E1 -10363.597,E2 -10363.597} C_VEL
LIN {X 0,Y 413.392,Z 344.388,A -85,B 0,C 180,E1 -10365.026,E2 -10365.026} C_VEL
LIN {X 0,Y 414.407,Z 333.689,A -85,B 0,C 180,E1 -10366.377,E2 -10366.377} C_VEL
LIN {X 0,Y 415.511,Z 321.829,A -85,B 0,C 180,E1 -10367.598,E2 -10367.598} C_VEL
LIN {X 0,Y 416.458,Z 310.172,A -85,B 0,C 180,E1 -10368.574,E2 -10368.574} C_VEL
LIN {X 0,Y 417.358,Z 296.662,A -85,B 0,C 180,E1 -10369.477,E2 -10369.477} C_VEL
LIN {X 0,Y 417.727,Z 288.387,A -85,B 0,C 180,E1 -10369.919,E2 -10369.919} C_VEL
LIN {X 0,Y 414.647,Z 274.806,A -85,B 0,C 180,E1 -10370.674,E2 -10370.674} C_VEL
LIN {X 0,Y 410.81,Z 261.27,A -85,B 0,C 180,E1 -10371.281,E2 -10371.281} C_VEL
LIN {X 0,Y 410.417,Z 259.386,A -85,B 0,C 180,E1 -10371.372,E2 -10371.372} C_VEL
LIN {X 0,Y 410.614,Z 254.485,A -85,B 0,C 180,E1 -10374.887,E2 -10374.887} C_VEL
LIN {X 0,Y 410.754,Z 249.42,A -85,B 0,C 180,E1 -10378.626,E2 -10378.626} C_VEL
LIN {X 0,Y 411.006,Z 245.044,A -85,B 0,C 180,E1 -10382.011,E2 -10382.011} C_VEL
LIN {X 0,Y 411.244,Z 240.66,A -85,B 0,C 180,E1 -10385.524,E2 -10385.524} C_VEL
LIN {X 0,Y 411.301,Z 237.456,A -85,B 0,C 180,E1 -10388.185,E2 -10388.185} C_VEL
LIN {X 0,Y 411.154,Z 234.902,A -85,B 0,C 180,E1 -10390.508,E2 -10390.508} C_VEL
LIN {X 0,Y 411.175,Z 234.896,A -85,B 0,C 180,E1 -10393.134,E2 -10393.134} C_VEL
LIN {X 0,Y 411.168,Z 234.896,A -85,B 0,C 180,E1 -10395.881,E2 -10395.881} C_VEL
LIN {X 0,Y 411.153,Z 234.896,A -85,B 0,C 180,E1 -10398.774,E2 -10398.774} C_VEL
LIN {X 0,Y 411.19,Z 234.889,A -85,B 0,C 180,E1 -10402.026,E2 -10402.026} C_VEL
LIN {X 0,Y 411.207,Z 234.889,A -85,B 0,C 180,E1 -10405.666,E2 -10405.666} C_VEL
LIN {X 0,Y 411.192,Z 234.893,A -85,B 0,C 180,E1 -10409.152,E2 -10409.152} C_VEL
LIN {X 0,Y 411.262,Z 234.884,A -85,B 0,C 180,E1 -10412.522,E2 -10412.522} C_VEL
LIN {X 0,Y 411.223,Z 234.887,A -85,B 0,C 180,E1 -10415.784,E2 -10415.784} C_VEL
LIN {X 0,Y 411.199,Z 234.893,A -85,B 0,C 180,E1 -10418.966,E2 -10418.966} C_VEL
LIN {X 0,Y 411.253,Z 234.884,A -85,B 0,C 180,E1 -10422.085,E2 -10422.085} C_VEL
LIN {X 0,Y 411.262,Z 234.881,A -85,B 0,C 180,E1 -10425.147,E2 -10425.147} C_VEL
LIN {X 0,Y 411.286,Z 234.878,A -85,B 0,C 180,E1 -10428.167,E2 -10428.167} C_VEL
LIN {X 0,Y 411.441,Z 234.86,A -85,B 0,C 180,E1 -10432.192,E2 -10432.192} C_VEL
LIN {X 0,Y 411.469,Z 234.854,A -85,B 0,C 180,E1 -10434.118,E2 -10434.118} C_VEL
LIN {X 0,Y 411.512,Z 234.85,A -85,B 0,C 180,E1 -10438.042,E2 -10438.042} C_VEL
LIN {X 0,Y 411.457,Z 234.856,A -85,B 0,C 180,E1 -10440.979,E2 -10440.979} C_VEL
LIN {X 0,Y 411.46,Z 234.856,A -85,B 0,C 180,E1 -10442.937,E2 -10442.937} C_VEL
LIN {X 0,Y 411.436,Z 234.859,A -85,B 0,C 180,E1 -10445.882,E2 -10445.882} C_VEL
LIN {X 0,Y 411.32,Z 234.874,A -85,B 0,C 180,E1 -10448.846,E2 -10448.846} C_VEL
LIN {X 0,Y 411.286,Z 234.878,A -85,B 0,C 180,E1 -10451.833,E2 -10451.833} C_VEL
LIN {X 0,Y 411.264,Z 234.884,A -85,B 0,C 180,E1 -10454.852,E2 -10454.852} C_VEL
LIN {X 0,Y 411.247,Z 234.887,A -85,B 0,C 180,E1 -10457.915,E2 -10457.915} C_VEL
LIN {X 0,Y 411.199,Z 234.891,A -85,B 0,C 180,E1 -10461.034,E2 -10461.034} C_VEL
LIN {X 0,Y 411.207,Z 234.891,A -85,B 0,C 180,E1 -10464.217,E2 -10464.217} C_VEL
LIN {X 0,Y 411.174,Z 234.895,A -85,B 0,C 180,E1 -10467.484,E2 -10467.484} C_VEL
LIN {X 0,Y 411.199,Z 234.889,A -85,B 0,C 180,E1 -10469.713,E2 -10469.713} C_VEL
LIN {X 0,Y 411.209,Z 234.887,A -85,B 0,C 180,E1 -10473.156,E2 -10473.156} C_VEL
LIN {X 0,Y 411.194,Z 234.892,A -85,B 0,C 180,E1 -10476.552,E2 -10476.552} C_VEL
LIN {X 0,Y 411.213,Z 234.888,A -85,B 0,C 180,E1 -10479.727,E2 -10479.727} C_VEL
LIN {X 0,Y 411.175,Z 234.898,A -85,B 0,C 180,E1 -10483.133,E2 -10483.133} C_VEL
LIN {X 0,Y 411.212,Z 234.992,A -85,B 0,C 180,E1 -10485.963,E2 -10485.963} C_VEL
LIN {X 0,Y 411.82,Z 238.837,A -85,B 0,C 180,E1 -10488.668,E2 -10488.668} C_VEL
LIN {X 0,Y 412.148,Z 242.16,A -85,B 0,C 180,E1 -10490.881,E2 -10490.881} C_VEL
LIN {X 0,Y 412.089,Z 246.077,A -85,B 0,C 180,E1 -10493.351,E2 -10493.351} C_VEL
LIN {X 0,Y 411.681,Z 251.98,A -85,B 0,C 180,E1 -10496.887,E2 -10496.887} C_VEL
LIN {X 0,Y 411.339,Z 257.894,A -85,B 0,C 180,E1 -10500.298,E2 -10500.298} C_VEL
LIN {X 0,Y 410.989,Z 263.741,A -85,B 0,C 180,E1 -10503.602,E2 -10503.602} C_VEL
LIN {X 0,Y 410.648,Z 269.573,A -85,B 0,C 180,E1 -10506.819,E2 -10506.819} C_VEL
LIN {X 0,Y 410.515,Z 273.02,A -85,B 0,C 180,E1 -10508.684,E2 -10508.684} C_VEL
LIN {X 0,Y 414.191,Z 288.453,A -85,B 0,C 180,E1 -10509.309,E2 -10509.309} C_VEL
LIN {X 0,Y 416.854,Z 302.577,A -85,B 0,C 180,E1 -10510.048,E2 -10510.048} C_VEL
LIN {X 0,Y 417.353,Z 307.231,A -85,B 0,C 180,E1 -10510.318,E2 -10510.318} C_VEL
LIN {X 0,Y 416.408,Z 320.982,A -85,B 0,C 180,E1 -10511.155,E2 -10511.155} C_VEL
LIN {X 0,Y 415.339,Z 333.647,A -85,B 0,C 180,E1 -10512.14,E2 -10512.14} C_VEL
LIN {X 0,Y 414.228,Z 346.224,A -85,B 0,C 180,E1 -10513.363,E2 -10513.363} C_VEL
LIN {X 0,Y 413.176,Z 357.43,A -85,B 0,C 180,E1 -10514.713,E2 -10514.713} C_VEL
LIN {X 0,Y 412.25,Z 367.482,A -85,B 0,C 180,E1 -10516.192,E2 -10516.192} C_VEL
LIN {X 0,Y 411.6,Z 375.834,A -85,B 0,C 180,E1 -10517.676,E2 -10517.676} C_VEL
LIN {X 0,Y 410.831,Z 383.817,A -85,B 0,C 180,E1 -10519.403,E2 -10519.403} C_VEL
LIN {X 0,Y 410.416,Z 390.249,A -85,B 0,C 180,E1 -10521.134,E2 -10521.134} C_VEL
LIN {X 0,Y 410.16,Z 395.952,A -85,B 0,C 180,E1 -10523.111,E2 -10523.111} C_VEL
LIN {X 0,Y 409.988,Z 400.089,A -85,B 0,C 180,E1 -10525.083,E2 -10525.083} C_VEL
LIN {X 0,Y 409.877,Z 402.791,A -85,B 0,C 180,E1 -10527.051,E2 -10527.051} C_VEL
LIN {X 0,Y 409.915,Z 404.131,A -85,B 0,C 180,E1 -10529.018,E2 -10529.018} C_VEL
LIN {X 0,Y 409.915,Z 404.13,A -85,B 0,C 180,E1 -10530.982,E2 -10530.982} C_VEL
LIN {X 0,Y 409.877,Z 402.789,A -85,B 0,C 180,E1 -10532.948,E2 -10532.948} C_VEL
LIN {X 0,Y 409.987,Z 400.085,A -85,B 0,C 180,E1 -10534.917,E2 -10534.917} C_VEL
LIN {X 0,Y 410.159,Z 395.94,A -85,B 0,C 180,E1 -10536.889,E2 -10536.889} C_VEL
LIN {X 0,Y 410.415,Z 390.231,A -85,B 0,C 180,E1 -10538.866,E2 -10538.866} C_VEL
LIN {X 0,Y 410.831,Z 383.797,A -85,B 0,C 180,E1 -10540.597,E2 -10540.597} C_VEL
LIN {X 0,Y 411.582,Z 375.808,A -85,B 0,C 180,E1 -10542.324,E2 -10542.324} C_VEL
LIN {X 0,Y 412.405,Z 365.923,A -85,B 0,C 180,E1 -10544.054,E2 -10544.054} C_VEL
LIN {X 0,Y 413.333,Z 355.486,A -85,B 0,C 180,E1 -10545.533,E2 -10545.533} C_VEL
LIN {X 0,Y 414.391,Z 343.818,A -85,B 0,C 180,E1 -10546.884,E2 -10546.884} C_VEL
LIN {X 0,Y 415.454,Z 332.154,A -85,B 0,C 180,E1 -10547.982,E2 -10547.982} C_VEL
LIN {X 0,Y 416.512,Z 319.785,A -85,B 0,C 180,E1 -10548.921,E2 -10548.921} C_VEL
LIN {X 0,Y 417.29,Z 307.106,A -85,B 0,C 180,E1 -10549.684,E2 -10549.684} C_VEL
LIN {X 0,Y 416.445,Z 300.258,A -85,B 0,C 180,E1 -10550.08,E2 -10550.08} C_VEL
LIN {X 0,Y 413.778,Z 286.63,A -85,B 0,C 180,E1 -10550.769,E2 -10550.769} C_VEL
LIN {X 0,Y 410.536,Z 272.975,A -85,B 0,C 180,E1 -10551.332,E2 -10551.332} C_VEL
LIN {X 0,Y 410.843,Z 266.329,A -85,B 0,C 180,E1 -10554.956,E2 -10554.956} C_VEL
LIN {X 0,Y 411.137,Z 261.782,A -85,B 0,C 180,E1 -10557.487,E2 -10557.487} C_VEL
LIN {X 0,Y 411.433,Z 255.892,A -85,B 0,C 180,E1 -10560.827,E2 -10560.827} C_VEL
LIN {X 0,Y 411.802,Z 249.981,A -85,B 0,C 180,E1 -10564.277,E2 -10564.277} C_VEL
LIN {X 0,Y 412.103,Z 245.932,A -85,B 0,C 180,E1 -10566.723,E2 -10566.723} C_VEL
